	0:  // ═══ IDLE ═══
		Develop_L2_Step := 0;
		IF L2_StartTrig.Q THEN
			Develop_L2_AcceptedSeq := Develop_L2_RequestSeq;
			Develop_L2_ActiveCode  := Develop_L2_ActionCode;
			Develop_L2_ErrorCode   := 0;
			Develop_L2_Retryable   := FALSE;
			// 所有 Develop 动作都需要目标缸号确定泵组, 先校验并派生
			targetTank := Expand_Target_Tank;
			IF (targetTank < 1) OR (targetTank > 8) THEN
				Develop_L2_ErrorCode    := 102;        // 缸号超范围
				Develop_L2_Retryable    := TRUE;
				Develop_L2_CompletedSeq := Develop_L2_AcceptedSeq;
				Develop_L2_State        := 30;         // REJECTED
			ELSIF (Develop_L2_ActionCode = 10) OR (Develop_L2_ActionCode = 20)
			      OR (Develop_L2_ActionCode = 30) OR (Develop_L2_ActionCode = 40) THEN
				// 派生泵组 (复用 legacy step 0 公式)
				targetGroup := (targetTank - 1) / 4 + 1;
				targetNum   := (targetTank - 1) MOD 4 + 1;
				Expand_Group  := targetGroup;
				Expand_Number := targetNum;
				// 复位 A 动作局部步进 (镜像本 POU 急停复位集合)
				清洗STEP := 0;
				润洗展缸STEP := 0;
				上液step := 0;
				初始化step := 0;
				泵初始化完成 := FALSE;
				润洗计数 := 0;
				上液计数 := 0;
				Develop_L2_SafeState := 0;
				Develop_L2_State := 10;                // RUNNING
			ELSIF Develop_L2_ActionCode = 50 THEN
				// drain: 前置缸必须处于 Developing(40)
				IF Tank_State[targetTank] = 40 THEN
					Tank_Drain_Enable[targetTank] := TRUE;
					Develop_L2_State := 10;            // RUNNING
				ELSE
					Develop_L2_ErrorCode    := 501;    // 缸非 Developing, 不可排液
					Develop_L2_Retryable    := TRUE;
					Develop_L2_CompletedSeq := Develop_L2_AcceptedSeq;
					Develop_L2_State        := 30;     // REJECTED
				END_IF
			ELSE
				Develop_L2_ErrorCode    := 101;        // 未知动作码
				Develop_L2_Retryable    := TRUE;
				Develop_L2_CompletedSeq := Develop_L2_AcceptedSeq;
				Develop_L2_State        := 30;         // REJECTED
			END_IF
		END_IF

	10: // ═══ RUNNING ═══
		CASE Develop_L2_ActiveCode OF
			10:  // 初始化 (目标泵组)
				A00_initialization_初始化();
				Develop_L2_Step := 初始化step;
				IF 泵初始化完成 THEN
					泵初始化完成 := FALSE;
					Develop_L2_SafeState    := 10;   // READY
					Develop_L2_CompletedSeq := Develop_L2_AcceptedSeq;
					Develop_L2_State        := 20;   // DONE
				END_IF
			20:  // 清洗管路
				A10_pipeline_cleaning_清洗管路();
				Develop_L2_Step := 清洗STEP;
				IF Expand_Group_clean_OK THEN
					Expand_Group_clean_OK := FALSE;
					Develop_L2_CompletedSeq := Develop_L2_AcceptedSeq;
					Develop_L2_State        := 20;   // DONE
				END_IF
			30:  // 润洗展缸 (目标缸)
				A20_clean_expand_润洗展缸();
				Develop_L2_Step := 润洗展缸STEP;
				IF Expand_Group_clean_OK THEN
					Expand_Group_clean_OK := FALSE;
					Develop_L2_CompletedSeq := Develop_L2_AcceptedSeq;
					Develop_L2_State        := 20;   // DONE
				END_IF
			40:  // 上液 (目标缸)
				IF (Expand_Group > 0) AND (Expand_Number > 0) THEN
					A40_up_liquid_上液();
				END_IF
				Develop_L2_Step := 上液step;
				IF Expand_up_liquid_OK THEN
					Expand_up_liquid_OK := FALSE;
					Develop_L2_CompletedSeq := Develop_L2_AcceptedSeq;
					Develop_L2_State        := 20;   // DONE
				END_IF
			50:  // 排液 (桥接 Tank_Drain 数组; A50/PRG_TankDrain 独立并行推进)
				Develop_L2_Step := Tank_State[targetTank];
				IF Tank_Drain_Done[targetTank] THEN
					Develop_L2_SafeState    := 10;   // READY (缸已排空待取板)
					Develop_L2_CompletedSeq := Develop_L2_AcceptedSeq;
					Develop_L2_State        := 20;   // DONE
				END_IF
		END_CASE

	20, 30, 40, 50:  // ═══ 终态 ═══
		IF (NOT Develop_L2_Start) OR Develop_L2_Reset THEN
			// drain 完成后回 IDLE 时撤除 Enable (Tank_State 由上位机写 0 释放)
			IF Develop_L2_ActiveCode = 50 THEN
				Tank_Drain_Enable[targetTank] := FALSE;
			END_IF
			Develop_L2_State := 0;
		END_IF

END_CASE
END_ACTION

ACTION A00_initialization_初始化:
R_TRIG[1](CLK:=%MX2005.5 , Q=> );  //泵空闲中
R_TRIG[2](CLK:=%MX2005.5 , Q=> );  //泵空闲中

CASE 初始化step OF
	0:
		润洗展缸STEP:=0;
		清洗STEP:=0;
		上液step:=0;
		放硅胶板step:=0;
		展开step:=0;
		expand_initialization_OK:=FALSE;
		Expand_Group_clean_OK:=FALSE;
		Expand_up_liquid_OK:=FALSE;
		Expand_silica_gel_plate_OK:=FALSE;
		展开工位允许放硅胶板:=FALSE;
		展开工位允许取硅胶板:=FALSE;
		展开工位机器人到达准备点:=FALSE;
		展开工位机器人放硅胶板完成:=FALSE;
		展开工位取硅胶板完成:=FALSE;
		展开工位允许放硅胶板1:=FALSE;
		CASE Expand_Group OF
			1:
				CASE Expand_Number OF
					1:
						展缸1气缸1手动:=FALSE;
						展缸1气缸1自动:=FALSE;
						展缸1进液电池阀1手动:=FALSE;
						展缸1进液电池阀1自动:=FALSE;
						展缸1排液电池阀1手动:=FALSE;
						展缸1排液电池阀1自动:=FALSE;
						展缸1吹气电池阀1手动:=FALSE;
						展缸1吹气电池阀1自动:=FALSE;
					2:
						展缸1气缸2手动:=FALSE;
						展缸1气缸2自动:=FALSE;
						展缸1进液电池阀2手动:=FALSE;
						展缸1进液电池阀2自动:=FALSE;
						展缸1排液电池阀2手动:=FALSE;
						展缸1排液电池阀2自动:=FALSE;
						展缸1吹气电池阀2手动:=FALSE;
						展缸1吹气电池阀2自动:=FALSE;	
					3:
						展缸1气缸3手动:=FALSE;
						展缸1气缸3自动:=FALSE;
						展缸1进液电池阀3手动:=FALSE;
						展缸1进液电池阀3自动:=FALSE;	
						展缸1排液电池阀3手动:=FALSE;
						展缸1排液电池阀3自动:=FALSE;
						展缸1吹气电池阀3手动:=FALSE;
						展缸1吹气电池阀3自动:=FALSE;	
					4:
						展缸1气缸4手动:=FALSE;
						展缸1气缸4自动:=FALSE;
						展缸1进液电池阀4手动:=FALSE;
						展缸1进液电池阀4自动:=FALSE;	
						展缸1排液电池阀4手动:=FALSE;
						展缸1排液电池阀4自动:=FALSE;
						展缸1吹气电池阀4手动:=FALSE;
						展缸1吹气电池阀4自动:=FALSE;	
				END_CASE
				IF %MW1300=0 AND 泵站位符=FALSE  THEN
					转发转存:='/1Z0,2,2R$R';     //泵初始化指令 
					%MW1300:=LEN(STR:= 转发转存);   //发送字节数
					泵站位符:=TRUE;
					初始化STEP:=10;
				END_IF
			2:
				CASE Expand_Number OF
					1:
						展缸2气缸1手动:=FALSE;
						展缸2气缸1自动:=FALSE;
						展缸2进液电池阀1手动:=FALSE;
						展缸2进液电池阀1自动:=FALSE;
						展缸2排液电池阀1手动:=FALSE;
						展缸2排液电池阀1自动:=FALSE;
						展缸2吹气电池阀1手动:=FALSE;
						展缸2吹气电池阀1自动:=FALSE;
					2:
						展缸2气缸2手动:=FALSE;
						展缸2气缸2自动:=FALSE;
						展缸2进液电池阀2手动:=FALSE;
						展缸2进液电池阀2自动:=FALSE;
						展缸2排液电池阀2手动:=FALSE;
						展缸2排液电池阀2自动:=FALSE;
						展缸2吹气电池阀2手动:=FALSE;
						展缸2吹气电池阀2自动:=FALSE;	
					3:
						展缸2气缸3手动:=FALSE;
						展缸2气缸3自动:=FALSE;
						展缸2进液电池阀3手动:=FALSE;
						展缸2进液电池阀3自动:=FALSE;	
						展缸2排液电池阀3手动:=FALSE;
						展缸2排液电池阀3自动:=FALSE;
						展缸2吹气电池阀3手动:=FALSE;
						展缸2吹气电池阀3自动:=FALSE;	
					4:
						展缸2气缸4手动:=FALSE;
						展缸2气缸4自动:=FALSE;
						展缸2进液电池阀4手动:=FALSE;
						展缸2进液电池阀4自动:=FALSE;	
						展缸2排液电池阀4手动:=FALSE;
						展缸2排液电池阀4自动:=FALSE;
						展缸2吹气电池阀4手动:=FALSE;
						展缸2吹气电池阀4自动:=FALSE;
				END_CASE 
				 IF %MW1300=0 AND 泵站位符=FALSE  THEN
					转发转存:='/2Z0,2,2R$R';     //泵初始化指令 
					%MW1300:=LEN(STR:= 转发转存);   //发送字节数
					泵站位符:=TRUE;
					初始化STEP:=10;
				END_IF
		END_CASE

		展开工位允许放硅胶板:=FALSE;
	
		
		
	10:
		CASE Expand_Group OF
			1:
				IF %MW1300=0 THEN
					转发转存:='/1Q$R';          //查询泵状态指令
					%MW1300:=LEN(STR:= 转发转存);
				END_IF
				
				
				IF R_TRIG[1].Q THEN
					泵初始化完成:=TRUE;
					泵站位符:=FALSE;
					初始化STEP:=0;
				END_IF
			2:
				IF %MW1300=0 THEN
					转发转存:='/2Q$R';          //查询泵状态指令
					%MW1300:=LEN(STR:= 转发转存);
				END_IF
				
				IF R_TRIG[2].Q THEN
					泵初始化完成:=TRUE;
					泵站位符:=FALSE;
					初始化STEP:=0;
				END_IF
		END_CASE
END_CASE
END_ACTION

ACTION A10_pipeline_cleaning_清洗管路:
TON[2](IN:=清洗STEP=10,PT:=T#1S);
TON_0(IN:=清洗STEP=20, PT:=T#3S , Q=> , ET=> );
R_TRIG[5](CLK:=%MX2005.5 , Q=> );  //泵空闲中
CASE 清洗STEP OF
	0 :
		大真空泵站位[10]:=TRUE;
		IF %MW1300=0 AND 泵站位符=FALSE  THEN
			转发转存:=Expand_forward_instructions; 
			%MW1300:=LEN(STR:= 转发转存);   //发送字节数
			泵站位符:=TRUE;
			清洗STEP:=10;
		END_IF
	10:
		//TON[2](IN:=TRUE,PT:=T#1S);
		IF %MW1300=0 AND TON[2].Q THEN
			CASE Expand_Group OF
				1:
					转发转存:='/1Q$R';          //查询泵状态指令
				2:
					转发转存:='/2Q$R';          //查询泵状态指令
			END_CASE
			%MW1300:=LEN(STR:= 转发转存);
		END_IF
		
		
		IF R_TRIG[5].Q THEN
			泵站位符:=FALSE;
			清洗STEP:=20;
		END_IF
	20:
		
		IF TON_0.Q THEN
			大真空泵站位[10]:=FALSE;
			转发转存:='';
			%MW1300:=128;
			Expand_Group_clean_OK:=TRUE;
			清洗STEP:=0;
		END_IF

		
END_CASE
END_ACTION

ACTION A20_clean_expand_润洗展缸:
TON[1](IN:=润洗展缸STEP=15,PT:=T#0.1S);
TON_1(IN:= 润洗展缸STEP=20  , PT:=T#5S , Q=> , ET=> );
TON_2(IN:=润洗展缸STEP=30, PT:=T#3S, Q=> , ET=> );
TON[4](IN:=润洗展缸STEP=40,PT:=T#30S);
TON[10](IN:=(Expand_Group=1 AND  展缸1溶剂废液检测传感器) OR (Expand_Group=2 AND  展缸2溶剂废液检测传感器),PT:=T#10S);
R_TRIG[3](CLK:=%MX2005.5 , Q=> );  //泵空闲中



CASE 润洗展缸STEP OF
	0 :
		润洗计数:=0;
		CASE Expand_Group OF
			1:
				CASE Expand_Number OF
					1:
						展缸1进液电池阀1自动:=TRUE;
						展缸1排液电池阀1自动:=TRUE;
						展缸1气缸1自动:=TRUE;
						润洗展缸STEP:=10;
					2:
						展缸1进液电池阀2自动:=TRUE;
						展缸1排液电池阀2自动:=TRUE;
						展缸1气缸2自动:=TRUE;
						润洗展缸STEP:=10;
					3:
						展缸1进液电池阀3自动:=TRUE;
						展缸1排液电池阀3自动:=TRUE;
						展缸1气缸3自动:=TRUE;
						润洗展缸STEP:=10;
					4:
						展缸1进液电池阀4自动:=TRUE;
						展缸1排液电池阀4自动:=TRUE;
						展缸1气缸4自动:=TRUE;
						润洗展缸STEP:=10;
				END_CASE
			
			2:
				CASE Expand_Number OF
					1:
						展缸2进液电池阀1自动:=TRUE;
						展缸2排液电池阀1自动:=TRUE;
						展缸2气缸1自动:=TRUE;
						润洗展缸STEP:=10;
					2:
						展缸2进液电池阀2自动:=TRUE;
						展缸2排液电池阀2自动:=TRUE;
						展缸2气缸2自动:=TRUE;
						润洗展缸STEP:=10;
					3:
						展缸2进液电池阀3自动:=TRUE;
						展缸2排液电池阀3自动:=TRUE;
						展缸2气缸3自动:=TRUE;
						润洗展缸STEP:=10;
					4:
						展缸2进液电池阀4自动:=TRUE;
						展缸2排液电池阀4自动:=TRUE;
						展缸2气缸4自动:=TRUE;
						润洗展缸STEP:=10;
				END_CASE
		END_CASE
	10:		
		IF %MW1300=0 AND 泵站位符=FALSE  THEN
			转发转存:=Expand_forward_instructions;   
			%MW1300:=LEN(STR:= 转发转存);   //发送字节数
			泵站位符:=TRUE;
			润洗展缸STEP:=15;
		END_IF
	15:
		
		IF %MW1300=0 AND TON[1].Q THEN
			CASE Expand_Group OF
				1:
					转发转存:='/1Q$R';           //查询泵状态指令
				2:
					转发转存:='/2Q$R';           //查询泵状态指令
			END_CASE
			%MW1300:=LEN(STR:= 转发转存);
		END_IF
		
		IF R_TRIG[3].Q THEN
			泵站位符:=FALSE;
			润洗计数:=润洗计数+1;
			IF 润洗计数>=Expand_rinse_count THEN
				润洗计数:=0;
				润洗展缸STEP:=20;
			ELSE
				润洗展缸STEP:=10;
			END_IF
			
		END_IF
		
	20:
		//TON_1(IN:= TRUE  , PT:=T#5S , Q=> , ET=> );
		IF TON_1.Q THEN
			转发转存:='';    
			%MW1300:=128;
			润洗展缸STEP:=30;
		END_IF
	30:
		//TON_2(IN:=TRUE, PT:=T#2S, Q=> , ET=> );
		IF TON_2.Q THEN
			大真空泵站位[9]:=TRUE;
			IF TON[10].Q THEN
				
				CASE Expand_Group OF
					1:
						CASE Expand_Number OF
							1:
								展缸1进液电池阀1自动:=FALSE;
								
								展缸1吹气电池阀1自动:=TRUE;
								
								
								润洗展缸STEP:=40;
							2:
								展缸1进液电池阀2自动:=FALSE;
								
								展缸1吹气电池阀2自动:=TRUE;
								
								
								润洗展缸STEP:=40;
							3:
								展缸1进液电池阀3自动:=FALSE;
								
								展缸1吹气电池阀3自动:=TRUE;
								
								
								润洗展缸STEP:=40;
							4:
								展缸1进液电池阀4自动:=FALSE;
								
								展缸1吹气电池阀4自动:=TRUE;
								
								润洗展缸STEP:=40;
						END_CASE
					
					2:
						CASE Expand_Number OF
							1:
								展缸2进液电池阀1自动:=FALSE;
								
								展缸2吹气电池阀1自动:=TRUE;
								
								润洗展缸STEP:=40;
							2:
								展缸2进液电池阀2自动:=FALSE;
								
								展缸2吹气电池阀2自动:=TRUE;
								
								润洗展缸STEP:=40;
							3:
								展缸2进液电池阀3自动:=FALSE;
								
								展缸2吹气电池阀3自动:=TRUE;
								
								润洗展缸STEP:=40;
							4:
								展缸2进液电池阀4自动:=FALSE;
								
								展缸2吹气电池阀4自动:=TRUE;
								润洗展缸STEP:=40;
						END_CASE
				END_CASE
			END_IF
		END_IF
	40:
		IF TON[4].Q THEN
			大真空泵站位[9]:=FALSE;
			CASE Expand_Group OF
				1:
					CASE Expand_Number OF
						1:
							展缸1排液电池阀1自动:=FALSE;
							展缸1吹气电池阀1自动:=FALSE;
							
							Expand_Group_clean_OK:=TRUE;
							润洗展缸STEP:=0;
						2:
							展缸1排液电池阀2自动:=FALSE;
							展缸1吹气电池阀2自动:=FALSE;
							
							Expand_Group_clean_OK:=TRUE;
							润洗展缸STEP:=0;
						3:
							展缸1排液电池阀3自动:=FALSE;
							展缸1吹气电池阀3自动:=FALSE;
							
							Expand_Group_clean_OK:=TRUE;
							润洗展缸STEP:=0;
						4:
							展缸1排液电池阀4自动:=FALSE;
							
							展缸1吹气电池阀4自动:=FALSE;
							Expand_Group_clean_OK:=TRUE;
							润洗展缸STEP:=0;
					END_CASE
				
				2:
					CASE Expand_Number OF
						1:
							展缸2排液电池阀1自动:=FALSE;
							展缸2吹气电池阀1自动:=FALSE;
							
							Expand_Group_clean_OK:=TRUE;
							润洗展缸STEP:=0;
						2:
							展缸2排液电池阀2自动:=FALSE;
							展缸2吹气电池阀2自动:=FALSE;
							
							Expand_Group_clean_OK:=TRUE;
							润洗展缸STEP:=0;
						3:
							展缸2排液电池阀2自动:=FALSE;
							展缸2吹气电池阀3自动:=FALSE;
							
							Expand_Group_clean_OK:=TRUE;
							润洗展缸STEP:=0;
						4:
							展缸2排液电池阀2自动:=FALSE;
							展缸2吹气电池阀4自动:=FALSE;
							
							Expand_Group_clean_OK:=TRUE;
							润洗展缸STEP:=0;
					END_CASE
			END_CASE
		END_IF
END_CASE
END_ACTION

ACTION A40_up_liquid_上液:
R_TRIG[6](CLK:=%MX2005.5 , Q=> );  //泵空闲中
TON[9](IN:=上液step=20,PT:=T#0.5S,);
IF Expand_Group>0 AND Expand_Number>0 THEN
	CASE 上液step OF
		0:
			CASE Expand_Group OF
				1:
					CASE Expand_Number OF
						1:
							展缸1进液电池阀1自动:=TRUE;
							上液step:=10;
						2:
							展缸1进液电池阀2自动:=TRUE;
							上液step:=10;
						3:
							展缸1进液电池阀3自动:=TRUE;
							上液step:=10;
						4:
							展缸1进液电池阀4自动:=TRUE;
							上液step:=10;
					END_CASE
				2:
					CASE Expand_Number OF
						1:
							展缸2进液电池阀1自动:=TRUE;
							上液step:=10;
						2:
							展缸2进液电池阀2自动:=TRUE;
							上液step:=10;
						3:
							展缸2进液电池阀3自动:=TRUE;
							上液step:=10;
						4:
							展缸2进液电池阀4自动:=TRUE;
							上液step:=10;
					END_CASE
			END_CASE
		10:
			IF %MW1300=0 AND 泵站位符=FALSE  THEN
				转发转存:=Expand_forward_instructions; 
				%MW1300:=LEN(STR:= 转发转存);   //发送字节数
				泵站位符:=TRUE;
				上液step:=20;
			END_IF
		20:
		
			IF %MW1300=0 AND TON[9].Q  THEN
				CASE Expand_Group OF
					 1:
						 转发转存:='/1Q$R';          //查询泵状态指令
					 2:
						 转发转存:='/2Q$R';          //查询泵状态指令
				END_CASE
				%MW1300:=LEN(STR:= 转发转存);
			END_IF
			
			
			IF R_TRIG[6].Q THEN
				泵站位符:=FALSE;
				转发转存:='';
				%MW1300:=128;
				上液计数:=上液计数+1;
				IF 上液计数>=Expand_up_liquid_count THEN
					上液计数:=0;
					CASE Expand_Group OF
						1:
							CASE Expand_Number OF
								1:
									展缸1进液电池阀1自动:=FALSE;
									;
								2:
									展缸1进液电池阀2自动:=FALSE;
									
								3:
									展缸1进液电池阀3自动:=FALSE;
									
								4:
									展缸1进液电池阀4自动:=FALSE;
									
							END_CASE
						2:
							CASE Expand_Number OF
								1:
									展缸2进液电池阀1自动:=FALSE;
									
								2:
									展缸2进液电池阀2自动:=FALSE;
									
								3:
									展缸2进液电池阀3自动:=FALSE;
									
								4:
									展缸2进液电池阀4自动:=FALSE;
									
							END_CASE
						END_CASE
					Expand_up_liquid_OK:=TRUE;
					上液step:=0;
				ELSE
					上液step:=10;
				END_IF
			END_IF	
    END_CASE	
END_IF
END_ACTION

ACTION A30_silica_gel_plate_放硅胶板:



CASE 放硅胶板step OF
	0:
		
		放硅胶板step:=10;
	10:
		展开工位允许放硅胶板1:=TRUE;
		IF 展开工位机器人到达准备点 THEN
			CASE Expand_Group OF
				1:
					CASE Expand_Number OF
						1:
							展缸1气缸1自动:=FALSE;
							IF 展缸1气缸1原点 THEN
								展开工位允许放硅胶板:=TRUE;
								ParameterList1:=1;
								放硅胶板step:=20;
							END_IF
							
						2:
							展缸1气缸2自动:=FALSE;
							IF 展缸1气缸2原点 THEN
								ParameterList1:=2;
								展开工位允许放硅胶板:=TRUE;
								放硅胶板step:=20;
							END_IF
						3:
							展缸1气缸3自动:=FALSE;
							IF 展缸1气缸3原点 THEN
								ParameterList1:=3;
								展开工位允许放硅胶板:=TRUE;
								放硅胶板step:=20;
							END_IF
						4:
							展缸1气缸4自动:=FALSE;
							IF 展缸1气缸4原点 THEN
								ParameterList1:=4;
								展开工位允许放硅胶板:=TRUE;
								放硅胶板step:=20;
							END_IF
					END_CASE
				2:
					CASE Expand_Number OF
						1:
							展缸2气缸1自动:=FALSE;
							IF 展缸2气缸1原点 THEN
								ParameterList1:=5;
								展开工位允许放硅胶板:=TRUE;
								放硅胶板step:=20;
							END_IF
						2:
							展缸2气缸2自动:=FALSE;
							IF 展缸2气缸2原点 THEN
								ParameterList1:=6;
								展开工位允许放硅胶板:=TRUE;
								放硅胶板step:=20;
							END_IF
						3:
							展缸2气缸3自动:=FALSE;
							IF 展缸2气缸3原点 THEN
								ParameterList1:=7;
								展开工位允许放硅胶板:=TRUE;
								放硅胶板step:=20;
							END_IF
						4:
							展缸2气缸4自动:=FALSE;
							IF 展缸2气缸4原点 THEN
								ParameterList1:=8;
								展开工位允许放硅胶板:=TRUE;
								放硅胶板step:=20;
							END_IF
					END_CASE
			END_CASE	
		END_IF
	20:
		IF 展开工位机器人放硅胶板完成 THEN
			展开工位允许放硅胶板:=FALSE;
			展开工位允许放硅胶板1:=FALSE;
			CASE Expand_Group OF
				1:
					CASE Expand_Number OF
						1:
							展缸1气缸1自动:=TRUE ;
							IF 展缸1气缸1动点 THEN
								放硅胶板step:=30;
							END_IF
							
						2:
							展缸1气缸2自动:=TRUE;
							IF 展缸1气缸2动点 THEN
								
								放硅胶板step:=30;
							END_IF
						3:
							展缸1气缸3自动:=TRUE;
							IF 展缸1气缸3动点 THEN
								
								放硅胶板step:=30;
							END_IF
						4:
							展缸1气缸4自动:=TRUE ;
							IF 展缸1气缸4动点 THEN
								
								放硅胶板step:=30;
							END_IF
					END_CASE
				2:
					CASE Expand_Number OF
						1:
							展缸2气缸1自动:=TRUE;
							IF 展缸2气缸1动点 THEN
								
								放硅胶板step:=30;
							END_IF
						2:
							展缸2气缸2自动:=TRUE ;
							IF 展缸2气缸2动点 THEN
								
								放硅胶板step:=30;
							END_IF
						3:
							展缸2气缸3自动:=TRUE;
							IF 展缸2气缸3动点 THEN
								
								放硅胶板step:=30;
							END_IF
						4:
							展缸2气缸4自动:=TRUE;
							IF 展缸2气缸4动点 THEN
								
								放硅胶板step:=30;
							END_IF
					END_CASE
			END_CASE	
		END_IF
	30:
		展开工位机器人放硅胶板完成:=FALSE;
		Expand_silica_gel_plate_OK:=TRUE;
		放硅胶板step:=0;
	
	
	

END_CASE
END_ACTION

END_PROGRAM

// Device/Application/40_Man/Robotic_Process_机器人流程
PROGRAM Robotic_Process_机器人流程
VAR
	RB_Control_0: FB_RB_Control;
	
	TON: TON;
	R_TRIG: ARRAY[1..2] OF R_TRIG;
END_VAR


R_TRIG[1](CLK:=collect_Old_Plate_Slot>0);
R_TRIG[2](CLK:=scrape_Old_Plate_Slot>0);
//机器人流程
IF MODE_State=1 THEN	
	IF R_TRIG[1].Q THEN
		收集瓶组站位符:=TRUE;
	END_IF
	IF R_TRIG[2].Q THEN
		收集器组站位符:=TRUE;
	END_IF

	CASE 机器人流程 OF
		0:
			IF Status=0 THEN
				IF 上样点样允许放硅胶板 THEN
					机器人流程:=10;
				ELSIF  上样点样允许取硅胶板 AND scrape_Step=0 AND NOT 刮板拍照工位站位符 THEN 
					机器人流程:=20;
				ELSIF 拍照工位允许取硅胶板去展开 AND (Expand_Step=0 OR Expand_Step=30) THEN
					机器人流程:=30;
				ELSIF 展开工位允许取硅胶板 AND scrape_Step=0 AND NOT 刮板拍照工位站位符 THEN       //刮板拍照空闲
					机器人流程:=40;
				ELSIF scrape_Fetch_Rack_Plate>0 AND NOT 刮板拍照暂存工位传感器 THEN 
					机器人流程:=70;
				ELSIF collect_Fetch_Rack_Plate>0 AND NOT 收集平台暂存工位传感器 THEN
					机器人流程:=60;
				ELSIF collect_Old_Plate_Slot>0 AND 收集平台暂存工位传感器 AND NOT 收集瓶组站位符  THEN
					机器人流程:=80;
				ELSIF scrape_Old_Plate_Slot>0 AND 刮板拍照暂存工位传感器 AND  NOT 收集器组站位符 THEN
					机器人流程:=90;
				ELSIF 拍照工位允许放收集器 AND 刮板拍照暂存工位传感器 AND scrape_Consume_Slot>0 THEN 
					机器人流程:=100;
				ELSIF 拍照工位允许取收集器 AND collect_Step=0 THEN           //收集工位空闲
					机器人流程:=110;
				ELSIF 收集工位允许放收集瓶 AND 收集平台暂存工位传感器 AND collect_Consume_Slot>0 THEN
					机器人流程:=120;
				ELSIF 收集工位允许取收集器 AND collect_Powder_Return_Slot>0 THEN
					机器人流程:=130;
				ELSIF 收集工位允许机器人取收集瓶放暂存工位 AND collect_Consume_Slot>0 THEN
					机器人流程:=140;
				ELSIF 拍照工位允许取硅胶板放废料区 THEN
					机器人流程:=50;
				END_IF
			END_IF
			

	
//	取升降机硅胶板放点样机构上

		10:                                                  
			ParameterList3:=1;                           //取1号吸盘工具
			A00_取放工具();
			IF 取工具完成 THEN
				取工具完成:=FALSE;
				ParameterList3:=0; 
				机器人流程:=11;
			END_IF
		11:
			A10_取升降机硅胶板();
			IF 取升降硅胶板完成 THEN
				取升降硅胶板完成:=FALSE;
				机器人流程:=12;		
			END_IF
		12:
			A15_放点样硅胶板();
			IF 放点样硅胶板完成 THEN
				FunctionID:=0;
				放点样硅胶板完成:=FALSE;
				机器人流程:=0;
			END_IF
			
				




//取点样硅胶板放拍照机构上
		20:
			ParameterList3:=1;                           //取1号吸盘工具
			A00_取放工具();
			IF 取工具完成 THEN
				取工具完成:=FALSE;
				机器人流程:=21;
			END_IF
		21:
			A20_取点样硅胶板();
			IF 取点样硅胶板完成 THEN
				
				机器人流程:=22;
			END_IF
		22:
			IF 拍照工位允许放硅胶板 THEN
				
				机器人流程:=23;
			END_IF
		23:
			A35_放拍照硅胶板();
			IF 放拍照硅胶板完成 THEN
				FunctionID:=0;
				放拍照硅胶板完成:=FALSE;
				机器人流程:=0;
			END_IF




//取拍照机构硅胶板放展缸
		30:
			ParameterList3:=1;                           //取1号吸盘工具
			A00_取放工具();
			IF 取工具完成 THEN
				取工具完成:=FALSE;
				机器人流程:=31;
			END_IF
		31:
			A32_取拍照硅胶板();
			IF 取拍照硅胶板完成 THEN
				
				机器人流程:=32;
			END_IF
		32:
			IF 展开工位允许放硅胶板1 THEN
				机器人流程:=33;
			END_IF
		33:
			A25_放展缸硅胶板();
			IF 展开工位机器人放硅胶板完成 THEN
				FunctionID:=0;
				机器人流程:=0;
			END_IF
				
				



//取展缸硅胶板到拍照刮取机构
		40:
			ParameterList3:=1;                           //取1号吸盘工具
			A00_取放工具();
			IF 取工具完成 THEN
				取工具完成:=FALSE;
				机器人流程:=41;
			END_IF
		41:
			A30_取展缸硅胶板();
			IF 取展缸硅胶板完成 THEN
				取展缸硅胶板完成:=FALSE;
				展开工位允许取硅胶板:=FALSE;
				机器人流程:=42;
			END_IF
		42:
			IF 拍照工位允许放硅胶板 THEN
				机器人流程:=43;
			END_IF
		43:
			A35_放拍照硅胶板();
			IF 放拍照硅胶板完成 THEN
				FunctionID:=0;
				放拍照硅胶板完成:=FALSE;
				机器人流程:=0;
			END_IF
			
			





//取拍照刮取硅胶板放到废料区
		50:
			ParameterList3:=1;                           //取1号吸盘工具
			A00_取放工具();
			IF 取工具完成 THEN
				取工具完成:=FALSE;
				机器人流程:=51;
			END_IF
		51:
			A32_取拍照硅胶板();
			IF 取拍照硅胶板完成 THEN
				取拍照硅胶板完成:=FALSE;
				机器人流程:=52;
			END_IF
		52:
			A65_放废料硅胶板();
			IF 取刮板硅胶板放废料区完成 THEN
				拍照工位允许取硅胶板放废料区:=FALSE;
				取刮板硅胶板放废料区完成:=FALSE;
				FunctionID:=0;
				
				机器人流程:=0;
			END_IF







//取收集瓶组到暂存工位
		60:
			ParameterList3:=2;            //取2号大夹持工具
			A00_取放工具();
			IF 取工具完成 THEN
				取工具完成:=FALSE;
				机器人流程:=61;
			END_IF
		61:
			A41_取收集瓶组放暂存工位();
			IF 取收集瓶组放暂存工位完成 THEN
				collect_Fetch_Rack_Plate:=0;
				FunctionID:=0;
				机器人流程:=0;
				取收集瓶组放暂存工位完成:=FALSE;
			END_IF
			
			





//取收集器组到暂存工位
		70:
			ParameterList3:=2;            //取2号大夹持工具
			A00_取放工具();
			IF 取工具完成 THEN
				取工具完成:=FALSE;
				机器人流程:=71;
			END_IF
		71:
			A40_取收集器组放暂存工位();
			IF 取收集器组放暂存工位完成 THEN
				scrape_Fetch_Rack_Plate:=0;
				FunctionID:=0;
				机器人流程:=0;
				取收集器组放暂存工位完成:=FALSE;
			END_IF
		
		
		
		
		
//取收集瓶暂存工位到仓库
		80:
			ParameterList3:=2;            //取2号大夹持工具
			A00_取放工具();
			IF 取工具完成 THEN
				取工具完成:=FALSE;
				机器人流程:=81;
			END_IF
		81:
			A71_取暂存收集瓶放仓库();
			IF 取暂存收集瓶组放仓库完成 THEN
				collect_Old_Plate_Slot:=0;
				FunctionID:=0;
				机器人流程:=0;
				取暂存收集瓶组放仓库完成:=FALSE;
			END_IF		
		
		
		
		
		
	
	
	


//取收集器暂存工位到仓库
		90:
			ParameterList3:=2;            //取2号大夹持工具
			A00_取放工具();
			IF 取工具完成 THEN
				取工具完成:=FALSE;
				机器人流程:=91;
			END_IF
		91:
			A70_取暂存收集器组放仓库();
			IF 取暂存收集器组放仓库完成 THEN
				scrape_Old_Plate_Slot:=0;
				FunctionID:=0;
				机器人流程:=0;
				取暂存收集器组放仓库完成:=FALSE;
			END_IF	







//取暂存收集器到刮取位
		100:
			ParameterList3:=3;                           //取3号小夹持工具
			A00_取放工具();
			IF 取工具完成 THEN
				取工具完成:=FALSE;
				机器人流程:=101;
			END_IF	
		101:
			A45_取暂存收集器放刮板位();
			IF 取暂存收集器放刮板位完成 THEN
				scrape_Consume_Slot:=0;
				FunctionID:=0;
				取暂存收集器放刮板位完成:=FALSE;
				机器人流程:=0;
			END_IF
			
			






//取刮板拍照收集器到收集工位
		110:
			ParameterList3:=3;                           //取3号小夹持工具
			A00_取放工具();
			IF 取工具完成 THEN
				取工具完成:=FALSE;
				机器人流程:=111;
			END_IF
		111:
			A55_取刮板收集器放到收集工位();
			IF 取刮板收集器放到收集工位完成 THEN
				FunctionID:=0;
				取刮板收集器放到收集工位完成:=FALSE;
				机器人流程:=0;
			END_IF
			
	
	
	
	
	
	
	
//取暂存收集瓶到收集工位	
		120:
			ParameterList3:=3;                           //取3号小夹持工具
			A00_取放工具();
			IF 取工具完成 THEN
				取工具完成:=FALSE;
				机器人流程:=121;
			END_IF
		121:
			A50_取暂存收集瓶放收集工位();
			IF 取暂存收集瓶放收集工位完成 THEN
				FunctionID:=0;
				取暂存收集瓶放收集工位完成:=FALSE;
				机器人流程:=0;
			END_IF
			
			






//取收集器到暂存工位
		130:
			ParameterList3:=3;                           //取3号小夹持工具
			A00_取放工具();
			IF 取工具完成 THEN
				取工具完成:=FALSE;
				机器人流程:=131;
			END_IF
		131:
			A60_取收集器放暂存工位();
			IF 取收集器放暂存工位完成 THEN
				collect_Powder_Return_Slot:=0;
				收集器组站位符:=FALSE;
				收集工位放收集器完成:=TRUE;
				FunctionID:=0;
				机器人流程:=0;
				取收集器放暂存工位完成:=FALSE;
			END_IF
			
			




//取收集瓶到暂存工位
		140:
			ParameterList3:=3;                           //取3号小夹持工具
			A00_取放工具();
			IF 取工具完成 THEN
				取工具完成:=FALSE;
				机器人流程:=141;
			END_IF
		141:
			A65_取收集瓶放暂存工位();
			IF 取收集瓶放暂存工位完成 THEN
				scrape_Consume_Slot:=0;
				收集瓶组站位符:=FALSE;
				FunctionID:=0;
				机器人流程:=0;
				取收集瓶放暂存工位完成:=FALSE;
			END_IF
			


    END_CASE
END_IF

ACTION A30_取展缸硅胶板:




CASE 取展缸硅胶板step OF
	0:
		地轨轴11YDATE.fAbsTarget:=HMI_地轨轴11Y.position[5];     //地轨去展开位
		地轨轴11YDATE.xMoveAbs:=TRUE;
		IF 地轨轴11YDATE.bAbMoveDone THEN
			地轨轴11YDATE.xMoveAbs:=FALSE;
			取展缸硅胶板step:=10;
		END_IF
	10:
		IF  ParameterList1>0 AND Status=0 THEN
			FunctionID:=5;                                  //取展缸硅胶板
			Execute:=1;
			取展缸硅胶板step:=20;
		END_IF
	20:
		IF RO_ParameterList1>0 AND Status=2 THEN                       //取硅胶板完成
			Execute:=0;
			取展缸硅胶板完成:=TRUE;
			取展缸硅胶板step:=0;
		END_IF
END_CASE
END_ACTION

ACTION A60_取收集器放暂存工位:


CASE 取收集器放暂存工位step OF
	0:
		地轨轴11YDATE.fAbsTarget:=HMI_地轨轴11Y.position[3];     //地轨去取收集组位置暂存位置
			地轨轴11YDATE.xMoveAbs:=TRUE;
			取收集器放暂存工位step:=5;
			
	5:
		IF 地轨轴11YDATE.bAbMoveDone  THEN
			地轨轴11YDATE.xMoveAbs:=FALSE;
			FunctionID:=12;  
			ParameterList8:=6;                               //放收集器回暂存工位
			Execute:=1;
			取收集器放暂存工位step:=10;
		END_IF
	10:
		IF RO_ParameterList8=6  THEN                       //放收集器回暂存工位完成
			收集工位机器人到达收集器位置:=TRUE;
			取收集器放暂存工位step:=30;
		END_IF
	30:
		IF 收集工位机器人取收集器放回暂存工位 THEN
			ParameterList8:=7;                               //机器人去取收集器
			ParameterList7:=collect_Powder_Return_Slot;
			收集工位机器人取收集器放回暂存工位:=FALSE;
			取收集器放暂存工位step:=40;
		END_IF
	40:
		IF RO_ParameterList8=7 AND Status=2 THEN                         //到达夹持位置
			Execute:=0;
			取收集器放暂存工位完成:=TRUE;
			取收集器放暂存工位step:=0;
		END_IF
END_CASE
END_ACTION

ACTION A00_取放工具:



CASE 取工具setp OF
	0:
		IF RO_ParameterList3=ParameterList3 THEN
			取工具完成:=TRUE;
			取工具setp:=0;
		ELSE
			取工具setp:=5;
		END_IF
	5:
		地轨轴11YDATE.fAbsTarget:=HMI_地轨轴11Y.position[4];     //地轨去取工具位置
		地轨轴11YDATE.xMoveAbs:=TRUE;
		IF 地轨轴11YDATE.bAbMoveDone THEN
			地轨轴11YDATE.xMoveAbs:=FALSE;
			FunctionID:=23;                              //取工具ID
			Execute:=1;                                  //机器人启动                        
			取工具setp:=10;
		END_IF
	10:
		IF RO_ParameterList3=ParameterList3 AND Status=2 THEN                               //取工具完成                                   
			Execute:=0;
			取工具完成:=TRUE;
			取工具setp:=0;
		END_IF
END_CASE
END_ACTION

ACTION A35_放拍照硅胶板:




CASE 放拍照硅胶板step OF
	0:
		地轨轴11YDATE.fAbsTarget:=HMI_地轨轴11Y.position[2];     //地轨去刮板拍照位
		地轨轴11YDATE.xMoveAbs:=TRUE;
		IF 地轨轴11YDATE.bAbMoveDone AND Status=0 THEN
				地轨轴11YDATE.xMoveAbs:=FALSE;
				FunctionID:=6;                              //放拍照硅胶板
				ParameterList5:=1;                           //放硅胶板到刮板拍照位
				Execute:=1;                                  //机器人启动                        
				放拍照硅胶板step:=10;
		END_IF
	10:
		IF RO_ParameterList5=1 AND Status=2 THEN              //放硅胶板完成
			Execute:=0; 
			ParameterList5:=0;
			拍照工位放硅胶板完成:=TRUE;
			放拍照硅胶板完成:=TRUE;
			放拍照硅胶板step:=0;
		END_IF
END_CASE
END_ACTION

ACTION A65_放废料硅胶板:



CASE 取刮板硅胶板放废料区step OF
	0:
		地轨轴11YDATE.fAbsTarget:=HMI_地轨轴11Y.position[1];     //地轨去上样点样位置
			地轨轴11YDATE.xMoveAbs:=TRUE;
			IF 地轨轴11YDATE.bAbMoveDone THEN
				地轨轴11YDATE.xMoveAbs:=FALSE;
				取刮板硅胶板放废料区step:=5;
            END_IF
	5:
		IF  升降下料伺服允许放料 AND  Status=0 THEN
			
			FunctionID:=8; 
			ParameterList4:=3;                                     //机器人放到废料区
			Execute:=1; 
			取刮板硅胶板放废料区step:=10;
		END_IF
	10:
		IF RO_ParameterList4=3 AND Status=2  THEN                               //机器人放废料区完成
			Execute:=0; 
			刮板拍照工位站位符:=FALSE;
			升降下料机器人放废料完成:=TRUE;
			取刮板硅胶板放废料区完成:=TRUE;
			取刮板硅胶板放废料区step:=0;
		END_IF
END_CASE
END_ACTION

ACTION A41_取收集瓶组放暂存工位:


CASE 取收集瓶组放暂存工位step OF
	0:
			地轨轴11YDATE.fAbsTarget:=HMI_地轨轴11Y.position[6];     //地轨去取收集组位置
			地轨轴11YDATE.xMoveAbs:=TRUE;
			溶液收集瓶定位自动:=FALSE;
			取收集瓶组放暂存工位step:=10;
	10:
		IF 地轨轴11YDATE.bAbMoveDone AND Status=0 THEN
				地轨轴11YDATE.xMoveAbs:=FALSE;
				FunctionID:=21;                              //取收集瓶组
				ParameterList6:=collect_Fetch_Rack_Plate+6;       //取收集瓶组坐标
				Execute:=1;                                  //机器人启动                        
				取收集瓶组放暂存工位step:=20;
			END_IF
	20:
		IF RO_ParameterList6=ParameterList6 AND Status=2 THEN             //取收集瓶组完成
			Execute:=0;
			地轨轴11YDATE.fAbsTarget:=HMI_地轨轴11Y.position[3];     //地轨去收集工位
			地轨轴11YDATE.xMoveAbs:=TRUE;
			取收集瓶组放暂存工位step:=30;
		END_IF
	30:
		IF 地轨轴11YDATE.bAbMoveDone AND Status=0 THEN
				地轨轴11YDATE.xMoveAbs:=FALSE;
				FunctionID:=22;                              //放收集瓶组
				ParameterList6:=14;                         //放收集瓶组
				Execute:=1;                                  //机器人启动                        
				取收集瓶组放暂存工位step:=40;
		END_IF
	40:
		IF RO_ParameterList6=14 AND Status=2 THEN                        //放收集瓶完成
			Execute:=0; 
			ParameterList6:=0;
			溶液收集瓶定位自动:=TRUE;
			取收集瓶组放暂存工位完成:=TRUE;
			取收集瓶组放暂存工位step:=0;
		END_IF
END_CASE
END_ACTION

ACTION A40_取收集器组放暂存工位:




CASE 取收集器组放暂存工位step OF
	0:
		地轨轴11YDATE.fAbsTarget:=HMI_地轨轴11Y.position[6];     //地轨去取收集组位置
		地轨轴11YDATE.xMoveAbs:=TRUE;
		取收集器组放暂存工位step:=10;
	
	10:
		IF 地轨轴11YDATE.bAbMoveDone  AND Status=0 THEN
				地轨轴11YDATE.xMoveAbs:=FALSE;
				FunctionID:=19;                              //取收集器组
				ParameterList6:=scrape_Fetch_Rack_Plate;       //取收集器组坐标
				Execute:=1;                                  //机器人启动                        
				取收集器组放暂存工位step:=20;
			END_IF
	20:
		IF RO_ParameterList6=ParameterList6 AND Status=2 THEN             //取收集器组完成
			Execute:=0;
			地轨轴11YDATE.fAbsTarget:=HMI_地轨轴11Y.position[3];     //地轨去收集
			地轨轴11YDATE.xMoveAbs:=TRUE;
			取收集器组放暂存工位step:=30;
		END_IF
	30:
		IF 地轨轴11YDATE.bAbMoveDone AND Status=0 THEN
				地轨轴11YDATE.xMoveAbs:=FALSE;
				FunctionID:=20;                              //放收集器组
				ParameterList6:=13;                         //取收集器组坐标
				Execute:=1;                                  //机器人启动                        
				取收集器组放暂存工位step:=40;
		END_IF
	40:
		IF RO_ParameterList6=13  AND Status=2 THEN                        //放收集器完成
			Execute:=0; 
			粉末收集器定位自动:=TRUE;
			取收集器组放暂存工位完成:=TRUE;
			取收集器组放暂存工位step:=0;
		END_IF
	
END_CASE
END_ACTION

ACTION A15_放点样硅胶板:



CASE 放点样硅胶板step OF
	0:	IF  Status=0 THEN
	  		ParameterList4:=0;
			FunctionID:=2;                         //放点样硅胶板
			ParameterList2:=1;                     //机器人放硅胶板
			Execute:=1;
			放点样硅胶板step:=10;
	  	END_IF
		
	10:
		IF RO_ParameterList2=1 AND Status=2 THEN         //机器人放硅胶板完成
			上样点样放硅胶板完成:=TRUE;
			Execute:=0;
			放点样硅胶板完成:=TRUE;
			放点样硅胶板step:=0;
		END_IF
END_CASE
END_ACTION

ACTION A55_取刮板收集器放到收集工位:



CASE 取刮板收集器放到收集工位step OF
	0:
		地轨轴11YDATE.fAbsTarget:=HMI_地轨轴11Y.position[2];     //地轨去取收集组位置暂存位置
			地轨轴11YDATE.xMoveAbs:=TRUE;
			取刮板收集器放到收集工位step:=1;
	1:
		IF 地轨轴11YDATE.bAbMoveDone AND 拍照工位允许取收集器 AND  Status=0 THEN
			地轨轴11YDATE.xMoveAbs:=FALSE;
			拍照工位机器人退出工位完成:=FALSE;
			FunctionID:=11;
			Execute:=1;
			ParameterList5:=4;                          //机器人去夹持工位
			取刮板收集器放到收集工位step:=10;
		END_IF
	10:
		IF RO_ParameterList5=4 THEN
			拍照工位机器人到达收集器夹持位:=TRUE;
			取刮板收集器放到收集工位step:=20;
		END_IF
	20:
		IF 拍照工位机器人退出 THEN
			
			拍照工位机器人到达收集器夹持位:=FALSE;
			ParameterList5:=5;                          //机器人退出工位
			取刮板收集器放到收集工位step:=30;
		END_IF
	30:
		IF RO_ParameterList5=5 THEN
			拍照工位机器人退出完成:=TRUE;
			Execute:=0;
			地轨轴11YDATE.fAbsTarget:=HMI_地轨轴11Y.position[3];     //地轨去收集工位
			地轨轴11YDATE.xMoveAbs:=TRUE;
			取刮板收集器放到收集工位step:=40;
		END_IF
	40:
		IF 地轨轴11YDATE.bAbMoveDone THEN
			地轨轴11YDATE.xMoveAbs:=FALSE;                     
			取刮板收集器放到收集工位step:=50;
		END_IF
	50:
		IF 收集工位允许放收集器 AND  Status=0 THEN
			FunctionID:=12;                             //放收集工位收集器
			ParameterList8:=1;                         //机器人放收集器到夹持工位
			Execute:=1;
			取刮板收集器放到收集工位step:=60;
		END_IF
	60:
		IF RO_ParameterList8=1 THEN
			
			收集工位放收集器到工位:=TRUE;
			取刮板收集器放到收集工位step:=70;
		END_IF
	70:
		IF 收集工位允许机器人退出工位 THEN
			ParameterList8:=2;                     //机器人退出工位
			取刮板收集器放到收集工位step:=80;
		END_IF
	80:
		IF RO_ParameterList8=2 AND Status=2 THEN                //机器人退出工位完成
			Execute:=0;
			收集工位机器人退出完成:=TRUE;
			收集工位放收集器到工位:=FALSE;
			取刮板收集器放到收集工位完成:=TRUE;
			取刮板收集器放到收集工位step:=0;
		END_IF
END_CASE
END_ACTION

ACTION A45_取暂存收集器放刮板位:


CASE 取暂存收集器放刮板位step OF
	0:
		IF RO_ParameterList3=3 THEN
			ParameterList3:=0;
			Execute:=0;
			地轨轴11YDATE.fAbsTarget:=HMI_地轨轴11Y.position[2];     //地轨去刮板拍照位
			地轨轴11YDATE.xMoveAbs:=TRUE;
			取暂存收集器放刮板位step:=10;
		END_IF
	10:
		IF 地轨轴11YDATE.bAbMoveDone THEN
			地轨轴11YDATE.xMoveAbs:=FALSE;                     
			取暂存收集器放刮板位step:=20;
		END_IF
	20:
		IF 拍照工位允许放收集器 AND Status=0 THEN
			FunctionID:=9;                              //取暂存收集器
			ParameterList7:=scrape_Consume_Slot;           //取收集器
			Execute:=1;
			取暂存收集器放刮板位step:=30;
		END_IF
	30:
		IF RO_ParameterList7=ParameterList7  THEN                   //取收集器完成
			Execute:=0;
			取暂存收集器放刮板位step:=40;
		END_IF
	40:
		IF Status=0 THEN
			FunctionID:=10;                             //放收集器
			ParameterList5:=2;                         //机器人放收集器到夹持工位
			Execute:=1;
			取暂存收集器放刮板位step:=45;
		END_IF
	45:
		IF RO_ParameterList5=2 THEN
			拍照工位机器人到达夹持位:=TRUE;
			取暂存收集器放刮板位step:=50;
		END_IF
	50:
		IF 拍照工位机器人退出工位 THEN
			ParameterList5:=3;                         //机器人退出工位
			拍照工位机器人到达夹持位:=FALSE;
			取暂存收集器放刮板位step:=60;
		END_IF
	60:
		IF RO_ParameterList5=3 AND Status=2 THEN                    //机器人退出工位完成
			Execute:=0;
			拍照工位机器人退出工位完成:=TRUE;
			取暂存收集器放刮板位完成:=TRUE;
			取暂存收集器放刮板位step:=0;
		END_IF	
	
	
	
	
END_CASE
END_ACTION

ACTION A20_取点样硅胶板:



CASE 取点样硅胶板step OF
	0:
		地轨轴11YDATE.fAbsTarget:=HMI_地轨轴11Y.position[1];     //地轨去上样点样位置
			地轨轴11YDATE.xMoveAbs:=TRUE;
			IF 地轨轴11YDATE.bAbMoveDone THEN
				地轨轴11YDATE.xMoveAbs:=FALSE; 
				取点样硅胶板step:=5;
			END_IF
	5:
		IF  Status=0 THEN    //上样点样完成，展开准备完成
			FunctionID:=3;                              //取点样硅胶板
			ParameterList2:=2;                          //取硅胶板参数
			Execute:=1;                                  //机器人启动                        
			取点样硅胶板step:=10;
		END_IF
	10:
		IF RO_ParameterList2=2 AND Status=2 THEN
			Execute:=0;
			ParameterList2:=0;
			上样点样允许取硅胶板:=FALSE;
			取点样硅胶板完成:=TRUE;
			取点样硅胶板step:=0;
		END_IF
END_CASE
END_ACTION

ACTION A25_放展缸硅胶板:



CASE 放展缸硅胶板step OF
	0:	
		地轨轴11YDATE.fAbsTarget:=HMI_地轨轴11Y.position[5];     //地轨去展开位
		地轨轴11YDATE.xMoveAbs:=TRUE;
		IF 地轨轴11YDATE.bAbMoveDone AND Status=0 THEN
			地轨轴11YDATE.xMoveAbs:=FALSE;
			展开工位机器人到达准备点:=TRUE;
			放展缸硅胶板step:=5;
		END_IF
	5:
		IF 展开工位允许放硅胶板 THEN
			FunctionID:=4;                              //放展缸硅胶板
			Execute:=1;                                  //机器人启动       
			展开工位机器人到达准备点:=FALSE;
			放展缸硅胶板step:=10;
		END_IF
			
	10:
		IF RO_ParameterList1>0 AND Status=2 THEN                       //放硅胶板完成
			展开工位机器人放硅胶板完成:=TRUE;
			FunctionID:=0;
			Execute:=0;
			放展缸硅胶板step:=0;
		END_IF
END_CASE
END_ACTION

ACTION A50_取暂存收集瓶放收集工位:




CASE 取暂存收集瓶放收集工位step OF
	0:
		地轨轴11YDATE.fAbsTarget:=HMI_地轨轴11Y.position[3];     //地轨去取收集组位置暂存位置
			地轨轴11YDATE.xMoveAbs:=TRUE;
			取暂存收集瓶放收集工位step:=1;
	1:
		IF 地轨轴11YDATE.bAbMoveDone AND Status=0 THEN
			地轨轴11YDATE.xMoveAbs:=FALSE;
			FunctionID:=13;                             //取收集瓶
			ParameterList9:=collect_Consume_Slot;           //取收集瓶参数
			Execute:=1;
			取暂存收集瓶放收集工位step:=5;
		END_IF
	5:
		IF RO_ParameterList9=ParameterList9 AND 收集工位允许放收集瓶 THEN        //取收集瓶完成
			Execute:=0;
			取暂存收集瓶放收集工位step:=6;
		END_IF
	6:
		IF Status=0 THEN
			FunctionID:=15;  
			ParameterList8:=3;
			Execute:=1;
			取暂存收集瓶放收集工位step:=10;
		END_IF
	10:
		IF RO_ParameterList8=3 AND Status=2 THEN
				Execute:=0;
			收集工位放收集瓶完成:=TRUE;
			取暂存收集瓶放收集工位完成:=TRUE;
			取暂存收集瓶放收集工位step:=0;
		END_IF
END_CASE
END_ACTION

ACTION A71_取暂存收集瓶放仓库:






CASE 取暂存收集瓶组放仓库step OF
	0:
		地轨轴11YDATE.fAbsTarget:=HMI_地轨轴11Y.position[3];     //地轨去取收集组位置暂存位置
		地轨轴11YDATE.xMoveAbs:=TRUE;
		溶液收集瓶定位自动:=FALSE;
		取暂存收集瓶组放仓库step:=10;
	10:
		IF 地轨轴11YDATE.bAbMoveDone AND  Status=0 THEN
			地轨轴11YDATE.xMoveAbs:=FALSE;
			FunctionID:=14;                              //放收集器/瓶到仓库
			ParameterList6:=16;                          //取暂存收集器组
			Execute:=1; 
			取暂存收集瓶组放仓库step:=20;
		END_IF
	20:
		IF RO_ParameterList6=16 AND Status=2 THEN                      //取完成
			Execute:=0; 
			地轨轴11YDATE.fAbsTarget:=HMI_地轨轴11Y.position[6];     //地轨去放收集组位置
			地轨轴11YDATE.xMoveAbs:=TRUE;
			取暂存收集瓶组放仓库step:=30;
		END_IF
	30:
		IF 地轨轴11YDATE.bAbMoveDone AND Status=0 THEN
			地轨轴11YDATE.xMoveAbs:=FALSE;
			ParameterList6:=collect_Old_Plate_Slot+6;               //取暂存收集瓶组
			Execute:=1; 
			取暂存收集瓶组放仓库step:=40;
		END_IF
	40:
		IF RO_ParameterList6=collect_Old_Plate_Slot+6  AND Status=2 THEN
			取暂存收集瓶组放仓库完成:=TRUE;
			Execute:=0; 
			取暂存收集瓶组放仓库step:=0;
		END_IF
END_CASE
END_ACTION

ACTION A65_取收集瓶放暂存工位:

CASE 取收集瓶放暂存工位step OF
	0:
		地轨轴11YDATE.fAbsTarget:=HMI_地轨轴11Y.position[3];     //地轨去取收集组位置暂存位置
			地轨轴11YDATE.xMoveAbs:=TRUE;
			取收集瓶放暂存工位step:=5;
	5:
		IF 地轨轴11YDATE.bAbMoveDone AND 收集工位允许机器人取收集瓶放暂存工位 THEN
			地轨轴11YDATE.xMoveAbs:=FALSE;
			收集工位放收集瓶完成:=FALSE;
			FunctionID:=12;
			ParameterList8:=4;                               //到收集工位取收集瓶
			Execute:=1;
			取收集瓶放暂存工位step:=6;
		END_IF
	6:
		
		IF  RO_ParameterList8=4 AND Status=2 THEN
			取收集瓶放暂存工位step:=10;
			收集工位机器人放收集瓶到暂存工位完成:=TRUE;
			Execute:=0;
		END_IF
	10:
		IF Status=0 THEN
			ParameterList8:=5;                               //放收集瓶到暂存工位
			Execute:=1;
			ParameterList9:=collect_Consume_Slot;
			取收集瓶放暂存工位step:=20;
		END_IF
	20:
		IF RO_ParameterList8=5 AND Status=2 THEN                         //放收集瓶到暂存工位完成
			Execute:=0;
			取收集瓶放暂存工位step:=0;
			取收集瓶放暂存工位完成:=TRUE;
		END_IF
END_CASE
END_ACTION

ACTION A10_取升降机硅胶板:


CASE 取升降硅胶板step OF
		0:
			地轨轴11YDATE.fAbsTarget:=HMI_地轨轴11Y.position[1];     //地轨去上样点样位置
			地轨轴11YDATE.xMoveAbs:=TRUE;
			IF 地轨轴11YDATE.bAbMoveDone THEN
				地轨轴11YDATE.xMoveAbs:=FALSE; 
				IF 升降上料伺服允许取料 AND Status=0 THEN
					FunctionID:=1;                              //取升降硅胶板ID
					ParameterList4:=1;                           //去升降机构位置
					Execute:=1;                                  //机器人启动 
					取升降硅胶板step:=10;
				END_IF
			END_IF
			
		10:
			IF RO_ParameterList4=1 THEN                   //机器人到位
				升降上料机器人已吸住物料:=TRUE;
				取升降硅胶板step:=15;
			END_IF
		15:
			IF 升降上料伺服下降完成  THEN
				ParameterList4:=2;                        //机器人取物料
				取升降硅胶板step:=20;
			END_IF
			
		20:
			IF RO_ParameterList4=2 AND Status=2 THEN                //机器人取物料完成
				ParameterList4:=0;
				Execute:=0;
				升降上料机器人取料完成:=TRUE;
				取升降硅胶板完成:=TRUE;
				取升降硅胶板step:=0;
			END_IF
END_CASE
END_ACTION

ACTION A70_取暂存收集器组放仓库:


CASE 取暂存收集器组放仓库step OF
	0:
		IF RO_ParameterList3=2 THEN
			Execute:=0; 
			地轨轴11YDATE.fAbsTarget:=HMI_地轨轴11Y.position[3];     //地轨去取收集组位置暂存位置
			地轨轴11YDATE.xMoveAbs:=TRUE;
			取暂存收集器组放仓库step:=10;
			粉末收集器定位自动:=FALSE;
		END_IF
	10:
		IF 地轨轴11YDATE.bAbMoveDone AND  Status=0 THEN
			地轨轴11YDATE.xMoveAbs:=FALSE;
			粉末收集器定位自动:=FALSE;
			溶液收集瓶定位自动:=FALSE;
			FunctionID:=14;                              //放收集器/瓶到仓库
			ParameterList6:=15;                          //取暂存收集器组
			Execute:=1; 
			取暂存收集器组放仓库step:=20;
		END_IF
	20:
		IF RO_ParameterList6=15 AND  Status=2 THEN                      //取完成
			Execute:=0; 
			地轨轴11YDATE.fAbsTarget:=HMI_地轨轴11Y.position[6];     //地轨去放收集组位置
			地轨轴11YDATE.xMoveAbs:=TRUE;
			取暂存收集器组放仓库step:=30;
		END_IF
	30:
		IF 地轨轴11YDATE.bAbMoveDone AND  Status=0 THEN
			地轨轴11YDATE.xMoveAbs:=FALSE;
			ParameterList6:=scrape_Old_Plate_Slot;               //取暂存收集器组
			Execute:=1;
			取暂存收集器组放仓库step:=40;
		END_IF
	40:
		IF RO_ParameterList6=scrape_Old_Plate_Slot AND Status=2 THEN
			Execute:=0;
			取暂存收集器组放仓库完成:=TRUE;
			取暂存收集器组放仓库step:=0;
		END_IF
	
END_CASE
END_ACTION

ACTION A32_取拍照硅胶板:
CASE 取拍照硅胶完step OF
	0:
		地轨轴11YDATE.fAbsTarget:=HMI_地轨轴11Y.position[2];     //地轨去刮板拍照位
		地轨轴11YDATE.xMoveAbs:=TRUE;
		IF 地轨轴11YDATE.bAbMoveDone THEN
				地轨轴11YDATE.xMoveAbs:=FALSE;
				取拍照硅胶完step:=5;
		END_IF
	5:		
		IF (拍照工位允许取硅胶板去展开 OR 拍照工位允许取硅胶板放废料区) AND Status=0 THEN    
			FunctionID:=6;                              
			ParameterList5:=6;                           //机器人取硅胶板
			Execute:=1;             
			拍照工位允许取硅胶板去展开 := FALSE;
			取拍照硅胶完step:=10;
		END_IF
	10:
		IF RO_ParameterList5=6 AND Status=2 THEN
			Execute:=0;
			ParameterList6:=0;
			取拍照硅胶板完成:=TRUE;
			取拍照硅胶完step:=0;
		IF 拍照工位允许取硅胶板放废料区 THEN
			拍照工位机器人取硅胶板完成 := TRUE;
		END_IF
		END_IF
END_CASE
END_ACTION

END_PROGRAM

// Device/Application/25_FB_功能块/FB_RB_Control
FUNCTION_BLOCK FB_RB_Control
VAR_INPUT
	StartCmd     : BOOL;
StopCmd      : BOOL;
PauseCmd     : BOOL;
Reset:BOOL;
RobotRunning : BOOL;
RobotStopped : BOOL;
RobotPaused  : BOOL;
RobotAlarm   : BOOL;
PowerOn:BOOL;
END_VAR
VAR_OUTPUT
	StartOut     : BOOL;
StopOut      : BOOL;
PauseOut     : BOOL;
ResetOut:BOOL;
StatusRun    : BOOL;
StatusStop   : BOOL;
StatusPause  : BOOL;
StatusAlarm  : BOOL;
PowerOnOut:BOOL;
END_VAR
VAR
	State        : INT := 0;   // 当前状态
END_VAR

(* ================= 报警优先 ================= *)
IF RobotAlarm THEN
    State := 4;
END_IF

CASE State OF

    (* -------- 0：空闲 -------- *)
    0:
        StartOut := FALSE;
        StopOut  := TRUE;
        PauseOut := FALSE;
		ResetOut:=FALSE;
        IF StartCmd AND NOT RobotAlarm THEN
            State := 1;
        END_IF

    (* -------- 1：运行 -------- *)
    1:
		IF NOT PowerOn THEN
			PowerOnOut:=TRUE;
		ELSE
			PowerOnOut:=FALSE;
		END_IF
		IF PowerOn THEN
			StartOut := TRUE;
			StopOut  := FALSE;
			PauseOut := FALSE;
		END_IF
        

        IF StopCmd THEN
            State := 3;
        ELSIF PauseCmd THEN
            State := 2;
        
        END_IF

    (* -------- 2：暂停 -------- *)
    2:
        PauseOut := TRUE;
		StartOut := FALSE ;
        StopOut  := FALSE;
        IF StopCmd THEN
            State := 3;
        ELSIF  StartCmd AND NOT RobotAlarm THEN
            State := 1;
        END_IF

    (* -------- 3：停止 -------- *)
    3:
        StartOut := FALSE;
        StopOut  := TRUE;
        PauseOut := FALSE;

        IF RobotStopped THEN
            State := 0;
        END_IF

    (* -------- 4：报警 -------- *)
    4:
        StartOut := FALSE;
        StopOut  := TRUE;
        PauseOut := FALSE;

        IF  Reset THEN
			ResetOut:=TRUE;
            State := 0;
        END_IF

END_CASE

(* ================= 状态输出 ================= *)
StatusRun   := (State = 1);
StatusPause := (State = 2);
StatusStop  := (State = 0) OR (State = 3);
StatusAlarm := (State = 4);

END_FUNCTION_BLOCK

// Device/Application/40_Man/Sample_point_sampling_上样点样
PROGRAM Sample_point_sampling_上样点样
VAR
	初始化step: INT;
	清洗step: INT;
	清洗计数: INT;
	上样准备step: INT;
	放硅胶板STEP: INT;
	吸收液体step: INT;
	TON_0: TON;
	TON_1: TON;
	点样step: INT;
	stepTimer           : TON;       // 步骤内通用定时器（调试期模拟，实机替换为FB完成信号）
    bubbleIndex         : INT;       // Step 20 气泡序列循环索引
    cleanCounter        : INT;       // Step 10 清洗循环计数器
	泵初始化完成: BOOL;
	R_TRIG: ARRAY[1..12] OF R_TRIG;
	N: INT;
	A: INT;
	TON: ARRAY[1..11] OF TON;
	打样伺服移动step: INT;
	
	L2_StartTrig : R_TRIG;            // Sampling_L2_Start 上升沿检测器
END_VAR

IF (Sampling_ControlMode = 1) AND (Sampling_L2_State = 10) THEN
	IF (NOT 急停) OR (MODE_State <> 1) THEN
		Sampling_L2_ErrorCode    := 401;       // 急停或模式切换中断
		Sampling_L2_SafeState    := 90;        // RECOVERY_REQUIRED
		Sampling_L2_Retryable    := FALSE;
		Sampling_L2_CompletedSeq := Sampling_L2_AcceptedSeq;
		Sampling_L2_State        := 50;        // INTERRUPTED
	END_IF
END_IF

IF Sampling_X_coordinate>0 THEN 
TON[11](IN:=NOT 上样料架检测1 OR NOT 上样料架检测2,PT:=T#3S);
	IF TON[11].Q THEN
		上样料架报警:=TRUE;
	END_IF
END_IF

// ── 1. 急停联锁（最高优先级）──
IF NOT 急停 THEN
    Sampling_Step  := 0;
    Sampling_Done  := FALSE;
    Sampling_Error := TRUE;
    Sampling_Busy  := FALSE;
	初始化step:=0;
	清洗step:=0;
	清洗计数:=0;
	上样准备step:=0;
	放硅胶板STEP:=0;
	吸收液体step:=0;
	打样伺服移动step:=0;
	泵初始化完成:=FALSE;
	N:=0;
	A:=0;
    stepTimer(IN := FALSE, PT := T#0S);
    RETURN;
END_IF

// ── 2. 复位脉冲（用于错误恢复 / 强制清状态）──
IF Sampling_Reset THEN
    Sampling_Step  := 0;
    Sampling_Done  := FALSE;
    Sampling_Error := FALSE;
    Sampling_Busy  := FALSE;
    stepTimer(IN := FALSE, PT := T#0S);
    cleanCounter := 0;
    bubbleIndex  := 0;
    RETURN;
END_IF

// ── 3. Enable=FALSE 时清 Done（次周期复位握手）──
IF NOT Sampling_Enable THEN
    Sampling_Done := FALSE;
END_IF

// ── 4. 派生 Sampling_Busy（写者唯一：本 POU 是唯一写者，禁止他处赋值）──
Sampling_Busy := (Sampling_Step >= 10)
              AND (Sampling_Step <= 80)
              AND (NOT Sampling_Done);

IF MODE_State=1 THEN
	IF Sampling_ControlMode = 0 THEN     // LEGACY (默认, 行为与今天完全一致)
		CASE Sampling_Step OF
			0:  // ═══ 空闲：等待 Enable 上升 ═══
				IF Sampling_Enable AND (NOT Sampling_Done) THEN
					Sampling_Step := 5;
					stepTimer(IN := FALSE, PT := T#0S);  // 复位定时器
				END_IF
			5:
					A00_initialization_初始化();
					IF Sampling_initialization_OK THEN
						Sampling_initialization_OK:=FALSE;
						Sampling_Step:=10;
					END_IF
			10: // ═══ 清洗（消费 Sampling_clean_instructions + Sampling_clean_count）═══
				A10_clean_清洗();
				IF Sampling_Cleaning_OK THEN
					stepTimer(IN := FALSE, PT := T#0S);
					Sampling_Cleaning_OK:=FALSE;
					Sampling_Step := 20;
				END_IF
	
			20: // ═══ 上样准备 ═══
					A30_Sample_preparation_上样准备();
					IF Sampling_preparation_OK THEN
						Sampling_preparation_OK:=FALSE;
						Sampling_Step:=30;
					END_IF
			 30: // ═══ 放硅胶板（机械臂+传感器自治）═══
				A20_Place_materials_放硅胶板();
				IF Sampling_Place_materials_OK THEN
					Sampling_Place_materials_OK:=FALSE;
					stepTimer(IN := FALSE, PT := T#0S);
					Sampling_Step := 40;
				END_IF	
	
			40: // ═══ 吸液（消费 Sampling_X/Y_coordinate + Sampling_aspirate_instructions）═══
				A40_absorb_liquid_吸收液体();
				IF Sampling_liquid_absorption THEN
					Sampling_liquid_absorption:=FALSE;
					stepTimer(IN := FALSE, PT := T#0S);
					Sampling_Step := 50;
				END_IF
			50: // ═══ 点样（消费 Sampling_dispense_instructions）═══
				A50_Spray_sample_点样();
				IF Sampling_Spray_sample_OK  THEN
					Sampling_Spray_sample_OK:=FALSE;
					Sampling_Step := 60;
					
				END_IF
			60:
				IF  取点样硅胶板完成 THEN
					取点样硅胶板完成:=FALSE;
					stepTimer(IN := FALSE, PT := T#0S);
					Sampling_Done := TRUE;
					Sampling_Busy := FALSE;
					Sampling_Step := 0;
				END_IF
		
			90: // ═══ 故障态：等待外部 Sampling_Reset 脉冲 ═══
				Sampling_Error := TRUE;   // 故障态本身不动作，仅等待顶部复位逻辑
		END_CASE	
	ELSE                                  // L2
		Sampling_L2_Dispatch();
	END_IF
END_IF

ACTION A20_Place_materials_放硅胶板:



	CASE 放硅胶板STEP OF
	 	0:
			点样轴7YDATE.fAbsTarget:=HMI_点样轴7Y.position[1];
			点样轴7YDATE.xMoveAbs:=TRUE;
			放硅胶板STEP:=10;
		10:
			IF 点样轴7YDATE.bAbMoveDone THEN
				上样点样允许放硅胶板:=TRUE;
				点样轴7YDATE.xMoveAbs:=FALSE;
				放硅胶板STEP:=20;
			END_IF
		20:
			IF 上样点样放硅胶板完成 THEN
				上样点样允许放硅胶板:=FALSE;
				上样点样放硅胶板完成:=FALSE;
				上样定位自动:=TRUE;
				Sampling_Place_materials_OK:=TRUE;
				放硅胶板STEP:=0;
			END_IF
		
		
	 END_CASE
END_ACTION

ACTION A30_Sample_preparation_上样准备:
TON[2](IN:=上样准备step=2,PT:=T#0.5S);
R_TRIG[3](CLK:=%MX2005.5 , Q=> );  //泵空闲中

CASE 上样准备step OF
	0:
		上样轴5Z轴DATE.fAbsTarget:=0;
		上样轴5Z轴DATE.xMoveAbs:=TRUE;
		IF 上样轴5Z轴DATE.bAbMoveDone THEN
			N:=1;
			上样轴5Z轴DATE.xMoveAbs:=FALSE ;
			上样准备step:=1;
		END_IF
		
	1:
	
		CASE N OF
			1,2:
				IF %MW1300=0 AND NOT 泵站位符 THEN
					泵站位符:=TRUE;
					转发转存:=Sampling_prep_instructions[N];    
					%MW1300:=LEN(STR:= 转发转存);   //发送字节数
					上样准备step:=2;
				END_IF
		END_CASE
		
	2:
		IF %MW1300=0 AND TON[2].Q THEN 
		转发转存:='/4Q$R';          //查询泵状态指令
		%MW1300:=LEN(STR:= 转发转存);
		END_IF
		
		IF R_TRIG[3].Q THEN
			泵站位符:=FALSE;
			N:=N+1;
			IF N>2 THEN
				
				Sampling_preparation_OK:=TRUE;
				N:=0;
				上样准备step:=0;
			ELSE
				上样准备step:=1;
			END_IF
			
		END_IF
END_CASE
END_ACTION

ACTION A00_initialization_初始化:





CASE 初始化step OF
	0 :
		上样定位手动:=FALSE;
		上样定位自动:=FALSE;
		上样点样三通电池阀手动:=FALSE;
		上样点样三通电池阀自动:=FALSE;
		上样吹气手动:=FALSE;
		上样吹气自动:=FALSE;
		打样瓶上料轴3YDATE.fAbsTarget:=0;
		点样轴6XDATE.fAbsTarget:=0;
		点样轴7YDATE.fAbsTarget:=0;
		上样轴4X轴DATE.fAbsTarget:=0;
		上样轴5Z轴DATE.fAbsTarget:=0;
		上样点样允许放硅胶板:=FALSE;
		点样轴7YDATE.xMoveAbs:=FALSE;
		点样轴6XDATE.xMoveAbs:=FALSE;
		上样轴5Z轴DATE.xMoveAbs:=FALSE;
		上样轴4X轴DATE.xMoveAbs:=FALSE;
		打样瓶上料轴3YDATE.xMoveAbs:=FALSE;
		Sampling_Spray_sample_OK:=FALSE;
		Sampling_liquid_absorption:=FALSE;
		Sampling_preparation_OK:=FALSE;
		上样点样允许取硅胶板:=FALSE;
		上样点样放硅胶板完成:=FALSE;
		大真空泵站位[11]:=FALSE;
		清洗计数:=0;
		清洗step:=0;
		放硅胶板STEP:=0;
		上样准备step:=0;
		吸收液体step:=0;
		点样step:=0;
		初始化step:=5;
	5:
		上样轴5Z轴DATE.fAbsTarget:=0;
		上样轴5Z轴DATE.xMoveAbs:=TRUE;
		IF 上样轴5Z轴DATE.bAbMoveDone THEN
			点样轴7YDATE.fAbsTarget:=0  ;  
			点样轴6XDATE.fAbsTarget:=0  ; 
			上样轴4X轴DATE.fAbsTarget:=0;          
			上样轴4X轴DATE.xMoveAbs:=TRUE;
			点样轴7YDATE.xMoveAbs:=TRUE;
			点样轴6XDATE.xMoveAbs:=TRUE;
			初始化step:=6;
		END_IF
	6:
		IF 上样轴4X轴DATE.bAbMoveDone AND 上样轴5Z轴DATE.bAbMoveDone AND 点样轴6XDATE.bAbMoveDone AND 点样轴7YDATE.bAbMoveDone THEN
			初始化step:=10;
			上样轴4X轴DATE.xMoveAbs:=FALSE;
			点样轴7YDATE.xMoveAbs:=FALSE;
			上样轴5Z轴DATE.xMoveAbs:=FALSE;
			点样轴6XDATE.xMoveAbs:=FALSE;
		END_IF
	10:
		IF %MW1300=0 AND NOT 泵站位符 THEN
			泵站位符:=TRUE;
			转发转存:='/4Z0,1,1R$R';     //泵初始化指令 
			%MW1300:=LEN(STR:= 转发转存);   //发送字节数
			初始化STEP:=20;
		END_IF
	20:
		IF %MW1300=0 THEN
			转发转存:='/4Q$R';          //查询泵状态指令
			%MW1300:=LEN(STR:= 转发转存);
		END_IF
		R_TRIG[1](CLK:=%MX2005.5 , Q=> );  //泵空闲中
		IF R_TRIG[1].Q THEN
			泵站位符:=FALSE;
			初始化STEP:=30;
		END_IF
	30:
		
		
			Sampling_initialization_OK:=TRUE;
			初始化step:=0;
		

END_CASE
END_ACTION

ACTION A50_Spray_sample_点样:
TON[4](IN:=点样step=20,PT:=T#0.5S);
TON[5](IN:=点样气泡传感器,PT:=T#5S);
TON[7](IN:=点样step=10,PT:=T#0.5S);
R_TRIG[10](CLK:=%MX2005.5 , Q=> );  //泵空闲中

CASE 点样step OF
	0:
		点样轴6XDATE.xMoveAbs:=FALSE;
		点样轴7YDATE.xMoveAbs:=FALSE;
		点样step:=1;
	1:
		点样轴6XDATE.fAbsTarget:=HMI_点样轴6X.position[2];        //起始位
		点样轴7YDATE.fAbsTarget:=HMI_点样轴7Y.position[2];         //起始位
		点样轴6XDATE.xMoveAbs:=TRUE;
		点样轴7YDATE.xMoveAbs:=TRUE;
		点样step:=5;
	5:
		IF 点样轴6XDATE.bAbMoveDone AND 点样轴7YDATE.bAbMoveDone THEN
			点样轴6XDATE.xMoveAbs:=FALSE;
			点样轴7YDATE.xMoveAbs:=FALSE;
			IF  %MW1300=0 AND NOT 泵站位符 THEN
				
				泵站位符:=TRUE;
				转发转存:=Sampling_dispense_instructions[1];
				%MW1300:=LEN(STR:= 转发转存);
				上样点样三通电池阀自动:=TRUE;
				点样step:=10;
			END_IF
		END_IF
	10:
		IF  %MW1300=0 AND TON[7].Q THEN                        
				转发转存:='/4Q$R';          //查询泵状态指令
				%MW1300:=LEN(STR:= 转发转存);
				
				IF R_TRIG[10].Q THEN
					泵站位符:=FALSE;
					
					点样step:=15;
				END_IF
		END_IF
	15:
		IF  %MW1300=0 AND NOT 泵站位符 THEN
			上样吹气自动:=TRUE;
			泵站位符:=TRUE;
			转发转存:=Sampling_dispense_instructions[2];
			%MW1300:=LEN(STR:= 转发转存);
			点样轴6XDATE.fAbsTarget:=HMI_点样轴6X.position[3];             //终点位
			点样轴6XDATE.xMoveAbs:=TRUE;
			点样step:=20;
		END_IF

	20:
		IF  %MW1300=0 AND TON[4].Q THEN                        
				转发转存:='/4Q$R';          //查询泵状态指令
				%MW1300:=LEN(STR:= 转发转存);
				
				IF R_TRIG[10].Q THEN
					泵站位符:=FALSE;
					上样点样三通电池阀自动:=FALSE;
					上样吹气自动:=FALSE;
				END_IF
		END_IF
		CASE 打样伺服移动step OF
			0:
				IF 点样轴6XDATE.bAbMoveDone THEN
					点样轴6XDATE.xMoveAbs:=FALSE;
					IF 泵站位符 THEN
						打样伺服移动step:=10;
					ELSE
						点样step:=30;
					END_IF
					
				END_IF
			10:
				点样轴6XDATE.fAbsTarget:=HMI_点样轴6X.position[2];        //起始位
				点样轴6XDATE.xMoveAbs:=TRUE;
				打样伺服移动step:=20;
			20:
				IF 点样轴6XDATE.bAbMoveDone THEN
					点样轴6XDATE.xMoveAbs:=FALSE;
					打样伺服移动step:=30;
				END_IF
			30:
				点样轴6XDATE.fAbsTarget:=HMI_点样轴6X.position[3];             //终点位
				点样轴6XDATE.xMoveAbs:=TRUE;
				打样伺服移动step:=0;
				
		END_CASE
		
	30:
		点样轴6XDATE.fAbsTarget:=HMI_点样轴6X.position[1];        //清洗位
		点样轴6XDATE.xMoveAbs:=TRUE;
		IF 点样轴6XDATE.bAbMoveDone THEN
			点样轴7YDATE.fAbsTarget:=HMI_点样轴7Y.position[1]; 
			点样轴7YDATE.xMoveAbs:=TRUE;
		
		点样step:=40;
		END_IF
		
	40:
		IF 点样轴7YDATE.bAbMoveDone  THEN
			点样轴6XDATE.xMoveAbs:=FALSE;
			点样轴7YDATE.xMoveAbs:=FALSE;
			上样定位自动:=FALSE;
			上样点样允许取硅胶板:=TRUE;
			Sampling_Spray_sample_OK:=TRUE;
			点样step:=0;
		END_IF
 END_CASE
END_ACTION

ACTION A40_absorb_liquid_吸收液体:
TON_0(IN:=吸收液体step=30, PT:=T#0.5S , Q=> , ET=> );
TON_1(IN:=NOT 点样气泡传感器, PT:=T#5S , Q=> , ET=> );
R_TRIG[10](CLK:=%MX2005.5 , Q=> );  //泵空闲中

IF Sampling_X_coordinate>0 AND  Sampling_Y_coordinate>0  THEN
	CASE 吸收液体step OF
		0:
			上样轴5Z轴DATE.fAbsTarget:=0;
			上样轴5Z轴DATE.xMoveAbs:=TRUE;
			IF 上样轴5Z轴DATE.bAbMoveDone THEN
				上样轴5Z轴DATE.xMoveAbs:=FALSE;
				上样轴4X轴DATE.fAbsTarget:=HMI_上样轴4X轴.position[Sampling_X_coordinate];
				打样瓶上料轴3YDATE.fAbsTarget:=HMI_打样瓶上料轴3Y.position[Sampling_Y_coordinate];
				上样轴4X轴DATE.xMoveAbs:=TRUE;
				打样瓶上料轴3YDATE.xMoveAbs:=TRUE;
				吸收液体step:=10;
			END_IF
		10:
			IF 上样轴4X轴DATE.bAbMoveDone AND 打样瓶上料轴3YDATE.bAbMoveDone THEN
				上样轴4X轴DATE.xMoveAbs:=FALSE;
				打样瓶上料轴3YDATE.xMoveAbs:=FALSE;
				上样轴5Z轴DATE.fAbsTarget:=HMI_上样轴5Z轴.position[2];
				上样轴5Z轴DATE.xMoveAbs:=TRUE;
				吸收液体step:=20;
			END_IF
		20:
			IF 上样轴5Z轴DATE.bAbMoveDone THEN
				上样轴5Z轴DATE.xMoveAbs:=FALSE;
				A:=1;
				吸收液体step:=25;
			END_IF
		25:
			CASE A OF
				1,2:
					IF  %MW1300=0 AND NOT 泵站位符 THEN
						转发转存:=Sampling_sample_instructions[A];   //吸收液体
						%MW1300:=LEN(STR:= 转发转存);
						泵站位符:=TRUE;
						吸收液体step:=30;
					END_IF
			END_CASE
					
		
		30:
			IF  %MW1300=0 AND TON_0.Q THEN                        
				转发转存:='/4Q$R';          //查询泵状态指令
				%MW1300:=LEN(STR:= 转发转存);
				
				IF R_TRIG[10].Q THEN
					泵站位符:=FALSE;
					A:=A+1;
					IF A>2 THEN
						A:=0;
						大真空泵站位[11]:=FALSE;
						吸收液体step:=40;
					ELSE
						吸收液体step:=25;
					END_IF
				END_IF
			END_IF

		40:
			上样轴5Z轴DATE.fAbsTarget:=0;
			上样轴5Z轴DATE.xMoveAbs:=TRUE;
			IF 上样轴5Z轴DATE.bAbMoveDone THEN
				上样轴5Z轴DATE.xMoveAbs:=FALSE;
				Sampling_liquid_absorption:=TRUE;
				吸收液体step:=0;
			END_IF

	END_CASE
END_IF
END_ACTION

ACTION Sampling_L2_Dispatch:
L2_StartTrig(CLK := Sampling_L2_Start);

CASE Sampling_L2_State OF

	0:  // ═══ IDLE: 等待 Start 上升沿 ═══
		Sampling_L2_Step := 0;
		IF L2_StartTrig.Q THEN
			// 锁存请求 (序号与动作码一并冻结, 防主机中途改写)
			Sampling_L2_AcceptedSeq := Sampling_L2_RequestSeq;
			Sampling_L2_ActiveCode  := Sampling_L2_ActionCode;
			Sampling_L2_ErrorCode   := 0;
			Sampling_L2_Retryable   := FALSE;
			IF (Sampling_L2_ActionCode = 10)
			   OR (Sampling_L2_ActionCode = 20)
			   OR (Sampling_L2_ActionCode = 60)
			   OR (Sampling_L2_ActionCode = 70) THEN
				// 复位所有 A 动作局部步进 (与本 POU 急停复位块同一集合)
				初始化step := 0;
				清洗step := 0;
				清洗计数 := 0;
				上样准备step := 0;
				放硅胶板STEP := 0;
				吸收液体step := 0;
				打样伺服移动step := 0;
				泵初始化完成 := FALSE;
				N := 0;
				A := 0;
				Sampling_L2_SafeState := 0;       // UNKNOWN (运行中)
				Sampling_L2_State := 10;           // RUNNING
			ELSE
				// 未知动作码 -> 接受前拒绝 (可重试)
				Sampling_L2_ErrorCode    := 101;
				Sampling_L2_Retryable    := TRUE;
				Sampling_L2_CompletedSeq := Sampling_L2_AcceptedSeq;
				Sampling_L2_State        := 30;    // REJECTED
			END_IF
		END_IF

	10: // ═══ RUNNING: 按 ActiveCode 调对应 A 动作, 监视其完成标志 ═══
		CASE Sampling_L2_ActiveCode OF
			10:  // 初始化
				A00_initialization_初始化();
				Sampling_L2_Step := 初始化step;
				IF Sampling_initialization_OK THEN
					Sampling_initialization_OK := FALSE;
					Sampling_L2_SafeState    := 10;   // READY
					Sampling_L2_CompletedSeq := Sampling_L2_AcceptedSeq;
					Sampling_L2_State        := 20;   // DONE
				END_IF
			20:  // 清洗
				A10_clean_清洗();
				Sampling_L2_Step := 清洗step;
				IF Sampling_Cleaning_OK THEN
					Sampling_Cleaning_OK := FALSE;
					Sampling_L2_CompletedSeq := Sampling_L2_AcceptedSeq;
					Sampling_L2_State        := 20;   // DONE
				END_IF
			60:  // 吸样
				A40_absorb_liquid_吸收液体();
				Sampling_L2_Step := 吸收液体step;
				IF Sampling_liquid_absorption THEN
					Sampling_liquid_absorption := FALSE;
					Sampling_L2_CompletedSeq := Sampling_L2_AcceptedSeq;
					Sampling_L2_State        := 20;   // DONE
				END_IF
			70:  // 点样
				A50_Spray_sample_点样();
				Sampling_L2_Step := 点样step;
				IF Sampling_Spray_sample_OK THEN
					Sampling_Spray_sample_OK := FALSE;
					Sampling_L2_CompletedSeq := Sampling_L2_AcceptedSeq;
					Sampling_L2_State        := 20;   // DONE
				END_IF
		END_CASE

	20, 30, 40, 50:  // ═══ 终态: 保持到 Start 落沿或 L2_Reset, 再回 IDLE ═══
		IF (NOT Sampling_L2_Start) OR Sampling_L2_Reset THEN
			Sampling_L2_State := 0;
		END_IF

END_CASE
END_ACTION

ACTION A10_clean_清洗:
TON[1](IN:=清洗step=20,PT:=T#0.5S);
TON[6](IN:=清洗step=40,PT:=T#0.5S);
TON[8](IN:=清洗step=26,PT:=T#0.5S);
R_TRIG[2](CLK:=%MX2005.5 , Q=> );  //泵空闲中
R_TRIG[11](CLK:=%MX2005.5 , Q=> );  //泵空闲中
R_TRIG[12](CLK:=%MX2005.5 , Q=> );  //泵空闲中

CASE 清洗step OF
	0 :
		点样轴6XDATE.xMoveAbs:=FALSE;
		上样轴4X轴DATE.xMoveAbs:=FALSE;
		上样轴5Z轴DATE.xMoveAbs:=FALSE;
		清洗step:=5;
	5:
		点样轴6XDATE.fAbsTarget:=HMI_点样轴6X.position[1];               //6X清洗位置赋值
		上样轴4X轴DATE.fAbsTarget:=HMI_上样轴4X轴.position[9];           //4X清洗位置赋值
		点样轴6XDATE.xMoveAbs:=TRUE;
		上样轴4X轴DATE.xMoveAbs:=TRUE;
		清洗计数:=0;
		清洗step:=6;
	6:
		IF 上样轴4X轴DATE.bAbMoveDone THEN
			上样轴4X轴DATE.xMoveAbs:=FALSE;
			上样轴5Z轴DATE.fAbsTarget:=HMI_上样轴5Z轴.position[1];
			上样轴5Z轴DATE.xMoveAbs:=TRUE;
			清洗step:=7;
		END_IF

	7:
		IF  上样轴5Z轴DATE.bAbMoveDone AND 点样轴6XDATE.bAbMoveDone THEN
			上样轴5Z轴DATE.xMoveAbs:=FALSE;
			点样轴6XDATE.xMoveAbs:=FALSE;
			IF Sampling_clean_count>0 THEN
				清洗step:=10;
			ELSE
				清洗step:=60;
			END_IF
			
		END_IF
	10:
		IF %MW1300=0 AND NOT 泵站位符 THEN
			泵站位符:=TRUE;
			转发转存:=Sampling_clean_instructions[1];    
			%MW1300:=LEN(STR:= 转发转存);   //发送字节数
			大真空泵站位[11]:=TRUE;
			上样点样三通电池阀自动:=TRUE;
			清洗step:=20;
		END_IF
	20:
		IF %MW1300=0 AND TON[1].Q THEN
		转发转存:='/4Q$R';          //查询泵状态指令
		%MW1300:=LEN(STR:= 转发转存);
		END_IF
		
		IF R_TRIG[2].Q THEN
			上样点样三通电池阀自动:=FALSE;
			泵站位符:=FALSE;
			清洗step:=24;
		END_IF
	24:
		IF %MW1300=0 AND NOT 泵站位符 THEN
			泵站位符:=TRUE;
			转发转存:=Sampling_clean_instructions[1];    
			%MW1300:=LEN(STR:= 转发转存);   //发送字节数
			清洗step:=26;
		END_IF
	26:
		IF %MW1300=0 AND TON[8].Q THEN
		转发转存:='/4Q$R';          //查询泵状态指令
		%MW1300:=LEN(STR:= 转发转存);
		END_IF
		
		IF R_TRIG[11].Q THEN
			
			泵站位符:=FALSE;
			清洗step:=30;
		END_IF
	30:
		IF %MW1300=0 AND NOT 泵站位符 THEN
			泵站位符:=TRUE;
			转发转存:=Sampling_clean_instructions[2];    
			%MW1300:=LEN(STR:= 转发转存);   //发送字节数
			
			清洗step:=40;
		END_IF
				
	40:
		IF %MW1300=0 AND TON[6].Q THEN
		转发转存:='/4Q$R';          //查询泵状态指令
		%MW1300:=LEN(STR:= 转发转存);
		END_IF
		
		IF R_TRIG[12].Q THEN
			泵站位符:=FALSE;
			清洗step:=50;
		END_IF
	50:
		清洗计数:=清洗计数+1;
		IF  Sampling_clean_count> 清洗计数 THEN                 
			转发转存:='';
			%MW1300:=128;
			清洗step:=10;
		ELSIF  Sampling_clean_count<= 清洗计数 THEN
			转发转存:='';
			%MW1300:=128;
			清洗计数:=0;
			Sampling_Cleaning_OK:=TRUE;
			清洗step:=0;
		END_IF	
		上样点样三通电池阀自动:=FALSE;
		
	60:
		大真空泵站位[11]:=FALSE;
		Sampling_Cleaning_OK:=TRUE;
		清洗step:=0;
END_CASE
END_ACTION

END_PROGRAM

// Device/Application/40_Man/Collection_process_收集流程
PROGRAM Collection_process_收集流程
VAR
	准备step: INT;
	收集step: INT;
	TON_0: TON;
	搬运step: INT;
	ton3s: TON;
	ton5s: TON;
	i: INT;
	stepTimer: TON;
	R_TRIG: ARRAY[1..5] OF R_TRIG;
	泵初始化完成: BOOL;
	初始化STEP: INT;
	ton: ARRAY[1..10] OF TON;
	L2_StartTrig : R_TRIG;            // Collect_L2_Start 上升沿检测器
	L2_SubStep   : INT;              // collect(20) 子序列步进 (0=准备 1=收集 2=搬运)
END_VAR

// TON自复位：Q变TRUE后IN立即变FALSE，下周期复位，形成循环脉冲
// ton3s(IN := bEnable AND NOT ton3s.Q, PT := T#3S);
// 
// Q脉冲时翻转输出（Q仅维持一个周期，无需上升沿检测）
// IF ton3s.Q THEN
//     bOutput := NOT bOutput;
// END_IF

IF (Collect_ControlMode = 1) AND (Collect_L2_State = 10) THEN
	IF (NOT 急停) OR (MODE_State <> 1) THEN
		Collect_L2_ErrorCode    := 401;
		Collect_L2_SafeState    := 90;
		Collect_L2_Retryable    := FALSE;
		Collect_L2_CompletedSeq := Collect_L2_AcceptedSeq;
		Collect_L2_State        := 50;     // INTERRUPTED
	END_IF
END_IF

// ── 1. 急停联锁（最高优先级）──
IF NOT 急停 THEN
    collect_Step  := 0;
    collect_Done  := FALSE;
    collect_Error := TRUE;
    collect_Busy  := FALSE;
	准备step:=0;
	收集step:=0;
	搬运step:=0;
	初始化STEP:=0;
	泵初始化完成:=FALSE;
    stepTimer(IN := FALSE, PT := T#0S);
    RETURN;
END_IF

// ── 2. 复位脉冲（用于错误恢复 / 强制清状态）──
IF collect_Reset THEN
    collect_Step  := 0;
    collect_Done  := FALSE;
    collect_Error := FALSE;
    collect_Busy  := FALSE;
    stepTimer(IN := FALSE, PT := T#0S);
    RETURN;
END_IF

// ── 3. Enable=FALSE 时清 Done（次周期复位握手）──
//    上位机收到 Done 后会拉低 collect_Enable，本段确保下一周期 Done 自动归零，
//    避免 Done 残留导致 step 0 误判。
IF NOT collect_Enable THEN
    collect_Done := FALSE;
END_IF

// ── 4. 派生 collect_Busy（写者唯一：本 POU 是唯一写者，禁止他处赋值）──
collect_Busy := (collect_Step >= 10)
                    AND (collect_Step <= 80)
                    AND (NOT collect_Done);

IF MODE_State=1 THEN
	IF Collect_ControlMode = 0 THEN       // LEGACY (默认)
		CASE collect_Step OF
			0 :                      // 空闲：等待 Enable 上升
				 IF collect_Enable AND (NOT collect_Done) THEN
					collect_Step := 5;
				 END_IF
			
			5:	
				A00_initialization_初始化();
				IF 收集平台下压气缸原点 AND 收集平台夹持气缸原点 AND 收集平台升降气缸原点 AND 收集平台推出气缸原点 AND 泵初始化完成 THEN
					collect_Step:=10;
					泵初始化完成:=FALSE;
				END_IF
				
				
					
			10:                    //就位
					A10_preparation_准备();
				IF collect_prepare_OK THEN
					collect_prepare_OK:=FALSE;
					collect_Step:=20;
				END_IF
				
				
				
			20:                    //收集    	
				A20_collect_收集();
				IF collect_OK THEN
					
					FOR i := 1 TO collect_count BY 1 DO
						;   // 占位：单次打液动作（实机替换为真实调用）
					END_FOR
					collect_OK:=FALSE;
					collect_Step:=30;
				END_IF
				
				
			30:                    //物料搬运
				A30_transport_物料搬运();
				 IF 收集工位放收集器完成 THEN
					 收集工位放收集器完成:=FALSE;
					collect_Done := TRUE;
					collect_Step:=0;
				 END_IF	
				 
				 
			90: // 故障：等待外部 collect_Reset 脉冲（已在顶部统一处理）
				collect_Error := TRUE;   // 故障态本身不动作，仅等待复位
		END_CASE
	ELSE                                   // L2
		Collect_L2_Dispatch();
	END_IF
END_IF

ACTION A20_collect_收集:
ton[1](IN:=收集step=10,PT:=T#0.5S);
ton[2](IN:=收集step=30,PT:=T#10S);
R_TRIG[5](CLK:=%MX2005.5 , Q=> );  //泵空闲中
CASE 收集step OF
	0 :
		IF collect_forward_instructions<>'' THEN
			收集进液自动:=TRUE;
			
			
		END_IF
		IF %MW1300=0 AND 泵站位符=FALSE  THEN
			转发转存:=collect_forward_instructions; 
			%MW1300:=LEN(STR:= 转发转存);   //发送字节数
			泵站位符:=TRUE;
			收集step:=10;
		END_IF
	10:
		IF %MW1300=0 AND ton[1].Q THEN
			转发转存:='/3Q$R';          //查询泵状态指令
			%MW1300:=LEN(STR:= 转发转存);
		END_IF
		
		
		IF R_TRIG[5].Q THEN
			泵站位符:=FALSE;
			收集step:=20;
		END_IF
	

	20:
		IF TRUE  THEN    //注射泵完成//
			转发转存:='';
			%MW300:=128;
			收集进液自动:=FALSE;
			收集排液自动:=TRUE;
			收集正压排液自动:=TRUE;
			收集计数:=收集计数+1;
			收集step:=30;
		END_IF
	30:
		IF ton[2].Q THEN
			TON_0(IN:=TRUE, PT:=T#5S , Q=> , ET=> );
			IF 收集计数>=collect_count AND TON_0.Q THEN
				收集计数:=0;
				收集step:=40;
			ELSE
				收集排液自动:=FALSE;
				收集正压排液自动:=FALSE;
				收集step:=0;
			END_IF
		END_IF
	40:
		
			收集排液自动:=FALSE;
			收集正压排液自动:=FALSE;
			collect_OK:=TRUE;
			收集step:=0;

		

		
END_CASE
END_ACTION

ACTION A00_initialization_初始化:
R_TRIG[1](CLK:=%MX2005.5 , Q=> );  //泵空闲中

//初始化流程
CASE 初始化STEP OF
	0:
		收集下压气缸手动:=FALSE;
		收集下压气缸自动:=FALSE;
		收集夹持气缸手动:=FALSE;
		收集夹持气缸自动:=FALSE;
		收集升降气缸手动:=FALSE;
		收集升降气缸自动:=FALSE;
		收集伸缩气缸手动:=FALSE;
		收集伸缩气缸自动:=FALSE;
		收集进液手动:=FALSE;
		收集进液自动:=FALSE;
		收集排液手动:=FALSE;
		收集排液自动:=FALSE;
		收集正压排液手动:=FALSE;
		收集正压排液自动:=FALSE;
		溶液收集瓶定位手动:=FALSE;
		收集工位允许放收集瓶:=FALSE;
		收集工位允许放收集器:=FALSE;
		收集工位允许机器人退出工位:=FALSE;
		收集工位允许机器人取收集瓶放暂存工位:=FALSE;
		收集工位允许取收集器:=FALSE;
		收集工位机器人取收集器放回暂存工位:=FALSE;
		
	
		收集工位放收集瓶完成:=FALSE;
		收集工位放收集器到工位:=FALSE;
	
		收集工位机器人退出完成:=FALSE;
		
		收集工位机器人放收集瓶到暂存工位完成:=FALSE;
		
		收集工位机器人到达收集器位置:=FALSE;

		collect_prepare_OK:=FALSE;
		collect_OK:=FALSE;
		收集工位放收集器完成:=FALSE;
		收集step:=0;
		准备step:=0;
		搬运step:=0;
		IF %MW1300=0 AND NOT 泵站位符 THEN
			泵站位符:=TRUE;
			转发转存:='/3Z0,2,2R$R';     //泵初始化指令 
			%MW1300:=LEN(STR:= 转发转存);   //发送字节数
			初始化STEP:=10;
		END_IF
	10:
		IF %MW1300=0 THEN
			转发转存:='/3Q$R';          //查询泵状态指令
			%MW1300:=LEN(STR:= 转发转存);
		END_IF
		
		IF R_TRIG[1].Q THEN
			泵站位符:=FALSE;
			泵初始化完成:=TRUE;
			初始化STEP:=0;
		END_IF
END_CASE
END_ACTION

ACTION Collect_L2_Dispatch:
// 功能:
//   收集 L2 统一动作通道派发器。仅在 MODE_State=1 且 Collect_ControlMode=1 时由
//   POU body 调用 (与 legacy CASE collect_Step 互斥, 单写者)。
L2_StartTrig(CLK := Collect_L2_Start);

CASE Collect_L2_State OF

	0:  // ═══ IDLE ═══
		Collect_L2_Step := 0;
		IF L2_StartTrig.Q THEN
			Collect_L2_AcceptedSeq := Collect_L2_RequestSeq;
			Collect_L2_ActiveCode  := Collect_L2_ActionCode;
			Collect_L2_ErrorCode   := 0;
			Collect_L2_Retryable   := FALSE;
			IF (Collect_L2_ActionCode = 10) OR (Collect_L2_ActionCode = 20) THEN
				// 复位 A 动作局部步进与子序列 (镜像本 POU 急停复位集合)
				准备step := 0;
				收集step := 0;
				搬运step := 0;
				初始化STEP := 0;
				泵初始化完成 := FALSE;
				L2_SubStep := 0;
				Collect_L2_SafeState := 0;
				Collect_L2_State := 10;            // RUNNING
			ELSE
				Collect_L2_ErrorCode    := 101;
				Collect_L2_Retryable    := TRUE;
				Collect_L2_CompletedSeq := Collect_L2_AcceptedSeq;
				Collect_L2_State        := 30;     // REJECTED
			END_IF
		END_IF

	10: // ═══ RUNNING ═══
		CASE Collect_L2_ActiveCode OF
			10:  // 初始化 (镜像 legacy step 5: A00 + 四气缸原点 + 泵初始化完成)
				A00_initialization_初始化();
				Collect_L2_Step := 初始化STEP;
				IF 收集平台下压气缸原点 AND 收集平台夹持气缸原点
				   AND 收集平台升降气缸原点 AND 收集平台推出气缸原点
				   AND 泵初始化完成 THEN
					泵初始化完成 := FALSE;
					Collect_L2_SafeState    := 10;   // READY
					Collect_L2_CompletedSeq := Collect_L2_AcceptedSeq;
					Collect_L2_State        := 20;   // DONE
				END_IF
			20:  // 收集 = 准备 -> 收集 -> 搬运 (镜像 legacy step 10->20->30)
				CASE L2_SubStep OF
					0:
						A10_preparation_准备();
						Collect_L2_Step := 准备step;
						IF collect_prepare_OK THEN
							collect_prepare_OK := FALSE;
							L2_SubStep := 1;
						END_IF
					1:
						A20_collect_收集();
						Collect_L2_Step := 100 + 收集step;
						IF collect_OK THEN
							collect_OK := FALSE;
							L2_SubStep := 2;
						END_IF
					2:
						A30_transport_物料搬运();
						Collect_L2_Step := 200 + 搬运step;
						IF 收集工位放收集器完成 THEN
							收集工位放收集器完成 := FALSE;
							Collect_L2_CompletedSeq := Collect_L2_AcceptedSeq;
							Collect_L2_State        := 20;   // DONE
						END_IF
				END_CASE
		END_CASE

	20, 30, 40, 50:  // ═══ 终态 ═══
		IF (NOT Collect_L2_Start) OR Collect_L2_Reset THEN
			Collect_L2_State := 0;
		END_IF

END_CASE
END_ACTION

ACTION A30_transport_物料搬运:


CASE 搬运step OF
	0 :                     //复位气缸
		收集下压气缸自动:=FALSE;
		
		搬运step:=5;
	5:
		IF 收集平台下压气缸原点 THEN
			收集升降气缸自动:=FALSE;
			搬运step:=10;
		END_IF
	10:                    //复位伸缩气缸
		IF 收集平台升降气缸原点 THEN
			收集伸缩气缸自动:=TRUE;
			搬运step:=20;
		END_IF
	20:                    //允许机器人收集瓶
		IF 收集平台推出气缸动点 THEN
			收集工位允许机器人取收集瓶放暂存工位:=TRUE;
			搬运step:=30;
		END_IF
	30:
		IF 收集工位机器人放收集瓶到暂存工位完成 THEN
			收集工位允许机器人取收集瓶放暂存工位:=FALSE;
			收集工位机器人放收集瓶到暂存工位完成:=FALSE;
			收集伸缩气缸自动:=FALSE;
			收集工位允许取收集器:=TRUE;
			搬运step:=40;
		END_IF
	40:
		IF 收集工位机器人到达收集器位置 THEN
				收集工位机器人到达收集器位置:=FALSE;
			收集夹持气缸自动:=FALSE;
			收集工位允许取收集器:=FALSE;
			搬运step:=50;
		END_IF
	50:
		IF 收集平台夹持气缸原点 THEN
			收集工位机器人取收集器放回暂存工位:=TRUE;
			搬运step:=60;
		END_IF
	60:
		 IF 收集工位放收集器完成 THEN
		 	搬运step:=0;
		 END_IF
		
		
		

END_CASE
END_ACTION

ACTION A10_preparation_准备:
//准备工作
CASE 准备step OF	
	0:
		IF 收集平台夹持气缸原点 AND 收集平台下压气缸原点 THEN
		收集工位允许放收集器:=TRUE;
		准备step:=10;
		END_IF
	10:
		IF 收集工位放收集器到工位 THEN
			收集夹持气缸自动:=TRUE;
			收集工位允许放收集器:=FALSE;
			准备step:=20;
		END_IF
	20:
		IF 收集平台夹持气缸动点 THEN
			收集工位允许机器人退出工位:=TRUE;
			准备step:=30;
		END_IF
		
	30:
		IF 收集工位机器人退出完成 THEN
			
			收集工位机器人退出完成:=FALSE;
			收集工位允许机器人退出工位:=FALSE;
			准备step:=40;
		END_IF
	40 :
		IF 收集平台推出气缸原点 AND NOT 收集平台瓶子有无传感器 THEN
			收集伸缩气缸自动:=TRUE;
			准备step:=50;
		END_IF
	50:
		IF 收集平台推出气缸动点 THEN
			收集工位允许放收集瓶:=TRUE;
			准备step:=60;
		END_IF
	60:
	    IF 收集工位放收集瓶完成 THEN
	    	收集工位允许放收集瓶:=FALSE;
			收集工位放收集瓶完成:=FALSE;
			收集伸缩气缸自动:=FALSE;
			准备step:=70;
	    END_IF
	70:
		IF 收集平台推出气缸原点 AND 收集平台瓶子有无传感器 THEN
			收集升降气缸自动:=TRUE;
			准备step:=80;
		ELSIF 收集平台推出气缸原点 AND NOT 收集平台瓶子有无传感器 THEN
			收集伸缩气缸自动:=FALSE;
			准备step:=40;
		END_IF

	80:
		IF 收集平台升降气缸动点  THEN
			收集下压气缸自动:=TRUE;
			collect_prepare_OK:=TRUE;
			准备step:=0;
		END_IF
		
END_CASE
END_ACTION

END_PROGRAM

// Device/Application/40_Man/initialization
PROGRAM initialization
VAR
END_VAR

上样轴4X轴DATE.bHomed:=FALSE;
上样轴5Z轴DATE.bHomed:=FALSE;

END_PROGRAM

// Device/Application/40_Man/Photo_scraper_拍照刮板
PROGRAM Photo_scraper_拍照刮板
VAR
	初始化step: INT;
	拍照step: INT;
	刮板收集step: INT;
	机器人取物料step: INT;
	TON_0: TON;
	stepTimer           : TON;       // 步骤内通用定时器（调试期模拟，实机替换为FB完成信号）
    confirmLatched      : BOOL;      // Confirm 上升沿检测：上一周期 Confirm 值
    confirmRisingEdge   : BOOL;      // Confirm 上升沿脉冲（单周期有效）
    phaseA_done_15      : BOOL;      // Step 15 送板完成标志（Phase A 门控）
    phaseA_done_20      : BOOL;      // Step 20 送板完成标志（Phase A 门控）
	k_pass: INT;
	g_plate_surface_z: REAL := 20.5;
	g_total_depth: REAL := 1.0;
	L2_StartTrig : R_TRIG;            // PhotoScrape_L2_Start 上升沿检测器
END_VAR

IF (PhotoScrape_ControlMode = 1) AND (PhotoScrape_L2_State = 10) THEN
	IF (NOT 急停) OR (MODE_State <> 1) THEN
		PhotoScrape_L2_ErrorCode    := 401;
		PhotoScrape_L2_SafeState    := 90;
		PhotoScrape_L2_Retryable    := FALSE;
		PhotoScrape_L2_CompletedSeq := PhotoScrape_L2_AcceptedSeq;
		PhotoScrape_L2_State        := 50;     // INTERRUPTED
	END_IF
END_IF

// ── 1. 急停联锁（最高优先级）──
IF NOT 急停 THEN
    scrape_Step  := 0;
    scrape_Done  := FALSE;
    scrape_Error := TRUE;
    scrape_Busy  := FALSE;
    confirmLatched  := FALSE;
    confirmRisingEdge := FALSE;
    phaseA_done_15  := FALSE;
    phaseA_done_20  := FALSE;
	刮板拍照真空自动:=FALSE;
	刮板拍照无刷电机自动:=FALSE;
    stepTimer(IN := FALSE, PT := T#0S);
    RETURN;
END_IF

// ── 2. 复位脉冲（用于错误恢复 / 强制清状态）──
// TODO【逻辑判断】实机复位时应额外执行：
//   - 清空刮板电机运动指令
//   - 复位相机触发状态
IF scrape_Reset THEN
    scrape_Step  := 0;
    scrape_Done  := FALSE;
    scrape_Error := FALSE;
    scrape_Busy  := FALSE;
    confirmLatched  := FALSE;
    confirmRisingEdge := FALSE;
    phaseA_done_15  := FALSE;
    phaseA_done_20  := FALSE;
	初始化step:=0;
	拍照step:=0;
	刮板收集step:=0;
	机器人取物料step:=0;
	 scrape_IsLast := FALSE;       // ★ 新增
	
    stepTimer(IN := FALSE, PT := T#0S);
    RETURN;
END_IF

// ── 3. Enable=FALSE 时清 Done（次周期复位握手）──
//    上位机收到 Done 后会拉低 scrape_Enable，本段确保下一周期 Done 自动归零，
//    避免 Done 残留导致 Step 0 误判。
IF NOT scrape_Enable THEN
    scrape_Done := FALSE;
END_IF

// ── 4. 派生 scrape_Busy（写者唯一：本 POU 是唯一写者，禁止他处赋值）──
scrape_Busy := (scrape_Step >= 10)
            AND (scrape_Step <= 80)
            AND (NOT scrape_Done);

// ── 5. Confirm 上升沿检测（Phase A 门控）──
IF scrape_Step=15 OR ((PhotoScrape_ControlMode=1) AND scrape_WaitConfirm) THEN
    confirmRisingEdge := scrape_Confirm AND (NOT confirmLatched);
    confirmLatched    := scrape_Confirm;
ELSE
    // Phase A 未完成 → 不更新 confirmLatched，保留 PC 早写的 Confirm=TRUE
    confirmRisingEdge := FALSE;
END_IF


// ── 6. 主状态机（刮板序列器，Step 15/20 乒乓握手 + PhotoMode 路由）──
IF MODE_State=1 THEN	
	IF PhotoScrape_ControlMode = 0 THEN   // LEGACY (默认)
		CASE scrape_Step OF
			0:  // ═══ 空闲：等待 Enable 上升 ═══
				IF scrape_Enable AND (NOT scrape_Done) THEN
					scrape_Step := 10;
					stepTimer(IN := FALSE, PT := T#0S);  // 复位定时器
				END_IF
			10:
				IF scrape_PhotoMode=2 THEN
					scrape_Step := 15;
				ELSE
					A00_initialization_初始化();
					IF Camera_scraper_initialization_OK THEN
						Camera_scraper_initialization_OK:=FALSE;
						scrape_Step := 15;
						拍照工位允许取硅胶板去展开 := FALSE;
					END_IF
				END_IF				
				
			 15: // ═══ before-photo（PhotoMode=1 时经此路径 — 点样后拍照乒乓等待）═══
				A10_Material_camera_拍照硅胶板();
				stepTimer(IN := FALSE, PT := T#0S);
				phaseA_done_15 := TRUE;  // 标记送板完成
				IF Photo_preparation_completed_OK THEN
					IF scrape_PhotoMode = 1 THEN    ///只拍照
						scrape_Step := 16;  // before-photo 模式：去 Step 15 拍照
						拍照工位允许取硅胶板去展开:=TRUE;
						刮板拍照定位气缸自动:=FALSE;
					ELSIF scrape_PhotoMode=2 OR scrape_PhotoMode=0 THEN
						scrape_Step := 20;  // 完整刮板模式：去 Step 20 拍照+视觉+刮取
						Photo_preparation_completed_OK:=FALSE;
					END_IF
					
					scrape_PhotoMode := 0;  // 消费后复位：路由决策完成后清除 PhotoMode/拍照+刮取
				END_IF
			16:
				IF 取拍照硅胶板完成 THEN
					Photo_preparation_completed_OK:=FALSE;
					取拍照硅胶板完成:=FALSE;
					scrape_Done := TRUE;
					scrape_Step := 0;
				END_IF
		
			20: // ═══ 刮取（消费 scrape_gcode_instructions，按 G-code 路径刮板）═══
				IF g_pass_count = 0 THEN
						scrape_Step := 40;
				ELSE
					
					A20_Scraper_collection_刮板收集();
					IF Scraper_collection_completed THEN
						刮板拍照工位站位符:=TRUE;
						scrape_gcode_instructions := '';  // 消费 G-code 指令
						Scraper_collection_completed:=FALSE;
						stepTimer(IN := FALSE, PT := T#0S);
						scrape_Step := 30;
					END_IF
				END_IF
			
			 30: // ═══ 机器人取粉末收集器 ═══
				A30_Robot_material_retrieval_机器人取粉末收集器();
				IF Robot_completes_material_retrieval THEN
					stepTimer(IN := FALSE, PT := T#0S);
					scrape_IsLast := FALSE;   // ★ 新增：消费型变量子步内归零
					scrape_Done := TRUE;
					scrape_Busy := FALSE;
					Robot_completes_material_retrieval:=FALSE;
					scrape_Step := 0;
				END_IF
	
			90: // ═══ 故障态：等待外部 scrape_Reset 脉冲 ═══
				scrape_Error := TRUE;   // 故障态本身不动作，仅等待顶部复位逻辑
						
		END_CASE
	ELSE
		PhotoScrape_L2_Dispatch();
	END_IF
END_IF

ACTION A00_initialization_初始化:





CASE 初始化step OF
	0:
		刮板拍照真空自动:=FALSE;
		刮板拍照真空手动:=FALSE;
		刮板拍照无刷电机手动:=FALSE;
		刮板拍照无刷电机自动:=FALSE;
		刮板拍照定位气缸手动:=FALSE;
		刮板拍照定位气缸自动:=FALSE;
		粉末收集器定位手动:=FALSE;
		粉末收集器定位自动:=FALSE;
		刮板拍照遮光气缸手动:=FALSE;
		刮板拍照遮光气缸自动:=FALSE;
		刮板拍照旋转气缸手动:=FALSE;
		刮板拍照旋转气缸自动:=FALSE;
		刮板拍照下压气缸手动:=FALSE;
		刮板拍照下压气缸自动:=FALSE;
		拍照工位允许放硅胶板:=FALSE;
		拍照工位允许放收集器:=FALSE;
		拍照工位机器人退出工位:=FALSE;
		拍照工位允许取收集器:=FALSE;
		拍照工位机器人退出:=FALSE;
		scrape_WaitConfirm := FALSE;
		 scrape_IsLast := FALSE;       // ★ 新增
		拍照工位放硅胶板完成 := FALSE;
		
		拍照工位机器人到达夹持位 := FALSE;
		
		拍照工位机器人退出工位完成 := FALSE;
	
		拍照工位机器人到达收集器夹持位 := FALSE;
		
		拍照工位机器人退出完成 := FALSE;
		拍照工位允许取硅胶板放废料区 := FALSE;
		拍照工位允许取硅胶板去展开 := FALSE;
		拍照工位机器人取硅胶板完成 := FALSE;
		拍照step:=0;
		机器人取物料step:=0;
		刮板收集step:=0;
		
		Camera_scraper_initialization_OK:=FALSE;
		Photo_preparation_completed_OK:=FALSE;
		Scraper_collection_completed:=FALSE;
		Robot_completes_material_retrieval:=FALSE;
		初始化step:=5;
	5:
		刮板轴10ZDATE.xMoveAbs:=FALSE;
		刮板轴9XDATE.xMoveAbs:=FALSE;
		拍照轴8YDATE.xMoveAbs:=FALSE;
		初始化step:=6;
	6:
		刮板轴10ZDATE.fAbsTarget:=0;
		刮板轴10ZDATE.xMoveAbs:=TRUE;
		IF 刮板轴10ZDATE.bAbMoveDone THEN
			刮板轴10ZDATE.xMoveAbs:=FALSE;
			初始化step:=10;
		END_IF
	10:
		刮板轴9XDATE.fAbsTarget:=335;
		刮板轴9XDATE.xMoveAbs:=TRUE;
		IF 刮板轴9XDATE.bAbMoveDone THEN
			刮板轴9XDATE.xMoveAbs:=FALSE;
			初始化step:=20;
		END_IF
	20:
		IF 刮板拍照遮光气缸上位 THEN
			拍照轴8YDATE.fAbsTarget:=0;
			拍照轴8YDATE.xMoveAbs:=TRUE;
			IF 拍照轴8YDATE.bAbMoveDone THEN
				拍照轴8YDATE.xMoveAbs:=FALSE;
				Camera_scraper_initialization_OK:=TRUE;
				初始化step:=0;
			END_IF	
		END_IF		
	
END_CASE
END_ACTION

ACTION A10_Material_camera_拍照硅胶板:



CASE 拍照step OF
	0:
		刮板轴9XDATE.fAbsTarget:=335;
		刮板轴9XDATE.xMoveAbs:=TRUE;
		IF 刮板轴9XDATE.bAbMoveDone THEN
			刮板轴9XDATE.xMoveAbs:=FALSE;
			IF scrape_PhotoMode=2 THEN
				scrape_WaitConfirm := TRUE;  // 标记送板完成
				拍照step:=10;
			ELSE
				拍照step:=1;
			END_IF
		END_IF
	
	1:
		拍照工位允许放硅胶板:=TRUE;
		IF 拍照工位放硅胶板完成 THEN
			拍照工位允许放硅胶板:=FALSE;
			拍照工位放硅胶板完成:=FALSE;
			刮板拍照定位气缸自动:=TRUE;
			IF scrape_PhotoMode=1 THEN
				拍照step:=30;
			ELSE 
				拍照step:=10;
			END_IF
			
		END_IF
	10:
		拍照工位允许放收集器:=TRUE;
		IF 拍照工位机器人到达夹持位 THEN
			拍照工位允许放收集器:=FALSE;
			刮板拍照下压气缸自动:=TRUE;
			拍照step:=20;
		END_IF
	20:
		TON_0(IN:=TRUE, PT:=T#1S , Q=> , ET=> );
		IF TON_0.Q THEN
			拍照工位机器人退出工位:=TRUE;
			IF 拍照工位机器人退出工位完成 THEN
				拍照工位机器人退出工位完成:=FALSE;
				拍照工位机器人退出工位:=FALSE;
				刮板拍照下压气缸自动:=TRUE;
				IF scrape_PhotoMode=2 THEN
					scrape_WaitConfirm := FALSE;
					Photo_preparation_completed_OK:=TRUE;
					拍照step:=0;
				ELSE
					拍照step:=30;
				END_IF
				
			END_IF
		END_IF
	30:
		IF 刮板拍照遮光气缸上位  THEN
			拍照轴8YDATE.fAbsTarget:=420;
			拍照轴8YDATE.xMoveAbs:=TRUE;
			IF 拍照轴8YDATE.bAbMoveDone THEN
				拍照轴8YDATE.xMoveAbs:=FALSE;
				刮板拍照遮光气缸自动:=TRUE;
				拍照step:=40;
			END_IF
		END_IF
		
	40:
		IF 刮板拍照遮光气缸下位 THEN
			scrape_WaitConfirm := TRUE;  // 标记送板完成
			
			拍照step:=50;
		END_IF
	50:
		IF confirmRisingEdge THEN
			刮板拍照遮光气缸自动:=FALSE;
			scrape_WaitConfirm := FALSE;
			拍照step:=60;
		END_IF
	60:
		IF 刮板拍照遮光气缸上位 THEN
			拍照轴8YDATE.fAbsTarget:=0;
			拍照轴8YDATE.xMoveAbs:=TRUE;
			IF 拍照轴8YDATE.bAbMoveDone THEN
				拍照轴8YDATE.xMoveAbs:=FALSE;
				Photo_preparation_completed_OK:=TRUE;
				拍照step:=0;
			END_IF
		END_IF
	
	
	
	
	
	
	
	
END_CASE
END_ACTION

ACTION PhotoScrape_L2_Dispatch:
// 功能:
//   拍照刮板 L2 统一动作通道派发器。仅在 MODE_State=1 且 PhotoScrape_ControlMode=1
//   时由 POU body 调用 (与 legacy CASE scrape_Step 互斥, 单写者)。
// 参数: 无。返回: 无 (经 PhotoScrape_L2_* 反馈)。
L2_StartTrig(CLK := PhotoScrape_L2_Start);

CASE PhotoScrape_L2_State OF

	0:  // ═══ IDLE ═══
		PhotoScrape_L2_Step := 0;
		IF L2_StartTrig.Q THEN
			PhotoScrape_L2_AcceptedSeq := PhotoScrape_L2_RequestSeq;
			PhotoScrape_L2_ActiveCode  := PhotoScrape_L2_ActionCode;
			PhotoScrape_L2_ErrorCode   := 0;
			PhotoScrape_L2_Retryable   := FALSE;
			IF (PhotoScrape_L2_ActionCode = 10)
			   OR (PhotoScrape_L2_ActionCode = 20)
			   OR (PhotoScrape_L2_ActionCode = 30) THEN
				// 复位 A 动作局部步进与乒乓门控 (镜像 scrape_Reset 块的内部复位)
				初始化step := 0;
				拍照step := 0;
				刮板收集step := 0;
				机器人取物料step := 0;
				confirmLatched := FALSE;
				confirmRisingEdge := FALSE;
				phaseA_done_15 := FALSE;
				phaseA_done_20 := FALSE;
				PhotoScrape_L2_SafeState := 0;
				PhotoScrape_L2_State := 10;        // RUNNING
			ELSE
				PhotoScrape_L2_ErrorCode    := 101;
				PhotoScrape_L2_Retryable    := TRUE;
				PhotoScrape_L2_CompletedSeq := PhotoScrape_L2_AcceptedSeq;
				PhotoScrape_L2_State        := 30; // REJECTED
			END_IF
		END_IF

	10: // ═══ RUNNING ═══
		CASE PhotoScrape_L2_ActiveCode OF
			10:  // 初始化
				A00_initialization_初始化();
				PhotoScrape_L2_Step := 初始化step;
				IF Camera_scraper_initialization_OK THEN
					Camera_scraper_initialization_OK := FALSE;
					PhotoScrape_L2_SafeState    := 10;   // READY
					PhotoScrape_L2_CompletedSeq := PhotoScrape_L2_AcceptedSeq;
					PhotoScrape_L2_State        := 20;   // DONE
				END_IF
			20:  // 拍照
				A10_Material_camera_拍照硅胶板();
				PhotoScrape_L2_Step := 拍照step;
				IF Photo_preparation_completed_OK THEN
					Photo_preparation_completed_OK := FALSE;
					PhotoScrape_L2_CompletedSeq := PhotoScrape_L2_AcceptedSeq;
					PhotoScrape_L2_State        := 20;   // DONE
				END_IF
			30:  // 刮取 (CNC G-code 副通道由主机驱动)
				IF g_pass_count <= 0 THEN
					// 空操作 (镜像 legacy: g_pass_count=0 跳过刮板, 视为成功完成)
					PhotoScrape_L2_CompletedSeq := PhotoScrape_L2_AcceptedSeq;
					PhotoScrape_L2_State        := 20;   // DONE
				ELSE
					A20_Scraper_collection_刮板收集();
					PhotoScrape_L2_Step := 刮板收集step;
					IF Scraper_collection_completed THEN
						Scraper_collection_completed := FALSE;
						刮板拍照工位站位符 := TRUE;            // 镜像 legacy step 20 收尾
						scrape_gcode_instructions := '';      // 消费 G-code 指令
						PhotoScrape_L2_CompletedSeq := PhotoScrape_L2_AcceptedSeq;
						PhotoScrape_L2_State        := 20;   // DONE
					END_IF
				END_IF
		END_CASE

	20, 30, 40, 50:  // ═══ 终态 ═══
		IF (NOT PhotoScrape_L2_Start) OR PhotoScrape_L2_Reset THEN
			PhotoScrape_L2_State := 0;
		END_IF

END_CASE
END_ACTION

ACTION A20_Scraper_collection_刮板收集:


CASE 刮板收集step OF
	0:
		刮板拍照真空自动:=TRUE;
		//刮板拍照无刷电机自动:=TRUE;
		
		// 首次进入：初始化 k 与首 pass 的 Z
		IF k_pass = 0 THEN
			
			k_pass := 1;
			g_pass_z := g_plate_surface_z + g_total_depth / INT_TO_LREAL(g_pass_count);
		END_IF
   
		// 触发 CNC：bExe 直接拉高，PLC 侧已有的 SMC pipeline 自动执行
		 CNC启动:= TRUE;
		刮板收集step:=10;
		// 单 pass 完成 → 推进或退出
		
	10:
		IF CNC完成 THEN
			IF k_pass >= g_pass_count THEN
				CNC启动 := FALSE;
				k_pass := 0;
				刮板收集step:=20;
			ELSE
				k_pass := k_pass + 1;
				g_pass_z := g_plate_surface_z
						  + INT_TO_LREAL(k_pass) * g_total_depth
						  / INT_TO_LREAL(g_pass_count);
				 //Z轴高度计算   安全高度+刮取次数*总需要刮取的高速/需要刮取的次数
				CNC启动 := FALSE;   // 下个扫描周期上面 bExe := TRUE 形成上升沿，pipeline 重跑
				刮板收集step:=0;
			END_IF
		END_IF

	20:
		  IF scrape_IsLast THEN
				拍照工位允许取硅胶板放废料区:=TRUE;   // ★ 仅最后一次刮取后才允许送废料
				scrape_IsLast:=FALSE;
				scrape_PhotoMode:=0;
		  END_IF
		刮板拍照定位气缸自动:=FALSE;
		刮板拍照真空自动:=FALSE;
		刮板拍照无刷电机自动:=FALSE;
		CNC启动:=FALSE;
		刮板拍照旋转气缸自动:=TRUE;
		Scraper_collection_completed:=TRUE;
		刮板收集step:=0;

END_CASE
END_ACTION

ACTION A30_Robot_material_retrieval_机器人取粉末收集器:




CASE 机器人取物料step OF
	0:
		拍照工位允许取收集器:=TRUE;
		IF 拍照工位机器人到达收集器夹持位 THEN
			拍照工位允许取收集器:=FALSE;
			刮板拍照下压气缸自动:=FALSE;
			机器人取物料step:=10;
		END_IF
	10:
		IF 刮板拍照下压气缸上位 THEN
			拍照工位机器人退出:=TRUE;
			机器人取物料step:=20;
		END_IF
	20:
		IF 拍照工位机器人退出完成 THEN
			拍照工位机器人退出:=FALSE;
			刮板拍照旋转气缸自动:=FALSE;
			拍照工位机器人退出完成:=FALSE;
			机器人取物料step:=30;
			IF scrape_IsLast THEN
				
				机器人取物料step:=30;                    // ★ 最后一次：去 step 30 清板
			ELSE
				Robot_completes_material_retrieval:=TRUE; // ★ 中间：直接 Done，不清板
				机器人取物料step:=0;
			END_IF
		END_IF
	30:
		IF 拍照工位机器人取硅胶板完成 THEN
			拍照工位允许取硅胶板放废料区:=FALSE;
			拍照工位机器人取硅胶板完成:=FALSE;
			Robot_completes_material_retrieval:=TRUE;
			机器人取物料step:=0;
		END_IF	
END_CASE
END_ACTION

END_PROGRAM

